RoboDK station: Additive-Manufacturing-and-Machining-with-ABB-IRB-120-3-0-6.rdk

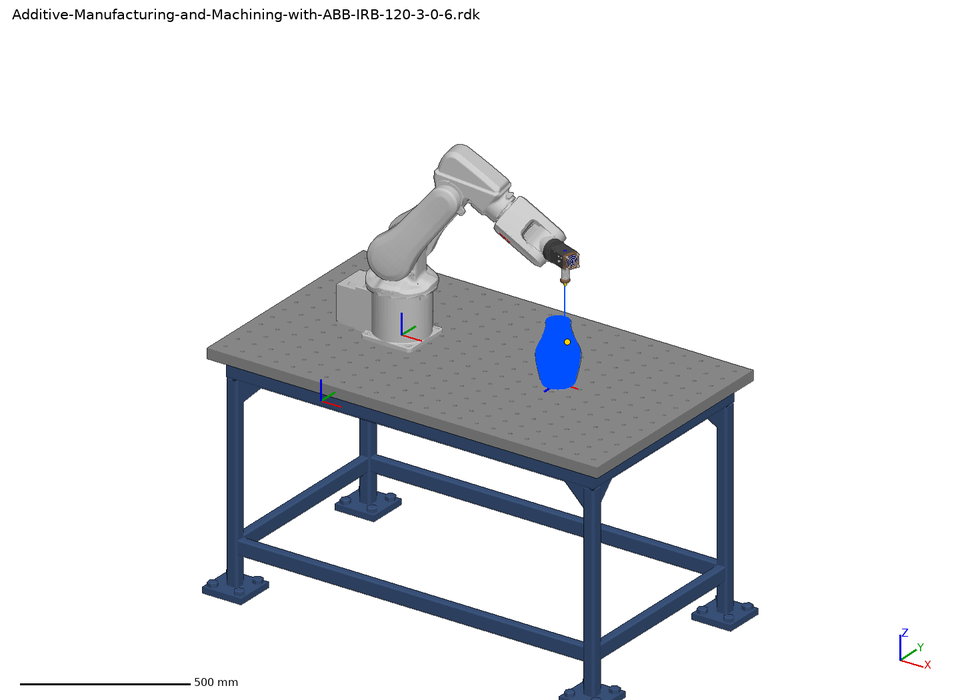
[picture v0: the station drawn from its stored meshes, robots at their saved joint values, targets as dots, program paths as lines]
Station Additive Manufacturing and Machining with ABB IRB 120-3/0.6 (saved by RoboDK 6.0.0). Poses are relative to the parent item; angles as X-Y-Z fixed-axis rotations.
Station parameters (name, value as stored): TAGS, ['Additive Manufacturing'], CEAD Extruder E40, 0
  - frame ABB IRB 120-3/0.6 Base at (-170, 0, 0) mm
    - robot ABB IRB 120-3/0.6: 6 axes, payload 3 kg, reach 580 mm, repeatability 0.01 mm, weight 25 kg
        modified DH rows (alpha deg, a mm, theta deg, d mm): 0, 0, 0, 290; -90, 0, -90, 0; 0, 270, 0, 0; -90, 70, 0, 302; 90, 0, 0, 0; -90, 0, 180, 72
        joint limits [-165, -110, -90, -160, -120, -400] to [165, 110, 70, 160, 120, 400]; home [0, 0, 0, 0, 0, 0]; saved at [10.704, 38.544, -4.293, -133.463, 44.707, 143.134]
      - tool ExtruderTool, TCP at (89.07, -8.14, 48.79) mm, rotated rx 0 ry 90 rz 0 deg, size 118.8 x 58.1 x 78.5 mm
    - object Table 1400x800x800mm at (-80, 0, 0) mm, size 1420 x 820 x 800 mm, geometry from UUID&
    - frame Part Reference at (560, 0, 0) mm, rotated rx 90 ry 0 rz 0 deg
      - object Simple Vase at (0, 0, 0) mm, size 135.9 x 200 x 135.9 mm, geometry from UUID&
      - frame NC File Frame at (-500, 0, 500) mm, rotated rx -90 ry 0 rz 0 deg
  - machining project Path1 settings: C:/Users/oli82/Desktop/List of demonstrations/8. G-code 3D printing/Vase.gcode | rotZ(0) | rotX(0)*rotY(0) | rotz(0)
  - program Path1 (30125 instructions, listed below)
  - Python program ExtrusionStart (listed below)
  - Python program ExtrusionStop (listed below)
  - notes Description: <!DOCTYPE HTML PUBLIC "-//W3C//DTD HTML 4.0//EN" "http://www.w3.org/TR/REC-html40/strict.dtd">
<html><head><meta name="qrichtext" content="1" /><style type="text/css">
p, li { white-space: pre-wrap; }
</style></head><body style=" font-family:'MS Shell Dlg 2'; font-size:8.25pt; font-weight:400; font-style:normal;">
<p style=" margin-top:0px; margin-bottom:0px; margin-left:0px; margin-right:0px; -qt-block-indent:0; text-indent:0px;">This example showcase the 3D printing of a vase using a ABB IRB 120-3/0.6 robot.<br /><br />Link for download : <a href="https://robodk.com/example/Additive-Manufacturing-and-Machining-with-ABB-IRB-120-3-0-6"><span style=" text-decoration: underline; color:#2a82da;">Additive Manufacturing and Machining with ABB IRB 120-3/0.6 robot | Examples Library</span></a></p></body></html>
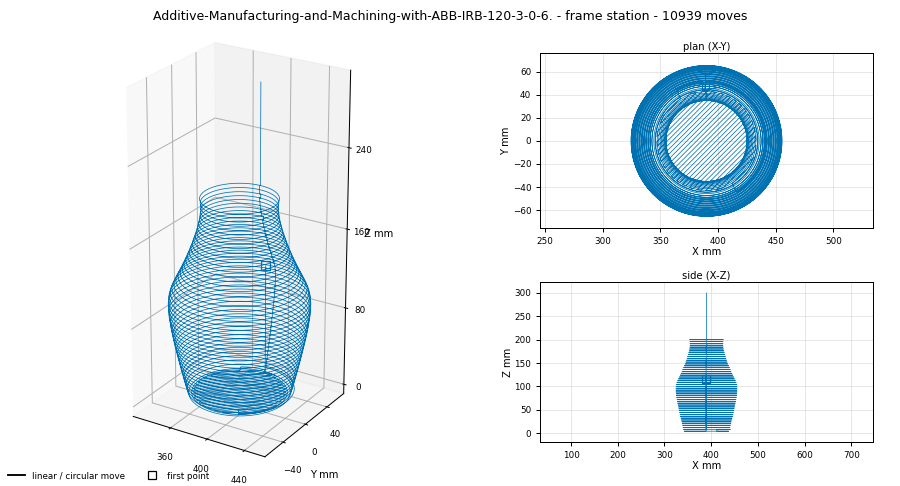
[picture p0: tool path of Additive-Manufacturing-and-Machining-with-ABB-IRB-120-3-0-6.rdk in frame station, 10939 of 10939 moves have a stored position in this frame; points joined in program order, loops and branches not executed]

--- program Path1 (robot ABB IRB 120-3/0.6) ---
  Smooth(1)
  Call SetRPM(200.0)
  Call M_RunCode(104)
  Call M_RunCode(105)
  Call SetRPM(200.0)
  Call M_RunCode(109)
  Call M_RunCode(82)
  Set speed (100.0 mm/s)
  Set speed (1000.0 mm/s)
  Set Ref.: NC File Frame
  Set Tool: ExtruderTool
  Show ExtruderTool
  MoveJ 1 to (499.11, 547.5, 115) mm, rotated rx 180 ry 0 rz 160 deg; joints [12.14, 61.149, -3.875, -143.247, 62.756, 161.126]
  MoveL 2 to (499.11, 547.5, 115) mm, rotated rx 180 ry 0 rz 160 deg; joints [12.14, 61.149, -3.875, -143.247, 62.756, 161.126]
  MoveL 3 to (499.11, 547.5, 15) mm, rotated rx -180 ry 0 rz 160 deg; joints [12.14, 78.131, -13.92, -145.093, 68.384, 165.584]
  Call ExtrusionStart
  MoveL 4 to (499.11, 547.5, 15) mm, rotated rx -180 ry 0 rz 160 deg; joints [12.14, 78.131, -13.92, -145.093, 68.384, 165.584]
  Call Extruder(0.00000)
  Set speed (3.3 mm/s)
  Call Extruder(3.00000)
  MoveL 5 to (499.11, 547.5, 15) mm, rotated rx -180 ry 0 rz 160 deg; joints [12.14, 78.131, -13.92, -145.093, 68.384, 165.584]
  Call Extruder(0.00000)
  Call Extruder(0.00000)
  Call Extruder(0.00000)
  Set speed (25.0 mm/s)
  Call Extruder(-6.50000)
  MoveL 6 to (499.11, 547.5, 15) mm, rotated rx -180 ry 0 rz 160 deg; joints [12.14, 78.131, -13.92, -145.093, 68.384, 165.584]
  Call M_RunCode(107)
  Set speed (60.0 mm/s)
  MoveL 7 to (499.11, 547.5, 4) mm, rotated rx 180 ry 0 rz 160 deg; joints [12.14, 80.192, -15.549, -145.19, 68.738, 165.849]
  Set speed (25.0 mm/s)
  Call Extruder(0.00000)
  MoveL 8 to (499.11, 547.5, 4) mm, rotated rx 180 ry 0 rz 160 deg; joints [12.14, 80.192, -15.549, -145.19, 68.738, 165.849]
  Set speed (30.0 mm/s)
  Call Extruder(3.94045)
  MoveL 9 to (497.01, 547.41, 4) mm, rotated rx 180 ry 0 rz 160 deg; joints [12.185, 79.885, -14.815, -145.238, 69.099, 166.093]
  Call Extruder(5.40756)
  MoveL 10 to (496.24, 547.36, 4) mm, rotated rx 180 ry 0 rz 160 deg; joints [12.199, 79.771, -14.543, -145.258, 69.233, 166.185]
  Call Extruder(7.73662)
  MoveL 11 to (495, 547.24, 4) mm, rotated rx -180 ry 0 rz 160 deg; joints [12.218, 79.591, -14.112, -145.292, 69.444, 166.331]
  Call Extruder(9.97998)
  MoveL 12 to (493.82, 547.1, 4) mm, rotated rx 180 ry 0 rz 160 deg; joints [12.232, 79.42, -13.698, -145.329, 69.647, 166.473]
  Call Extruder(11.58516)
  MoveL 13 to (492.97, 546.98, 4) mm, rotated rx 180 ry 0 rz 160 deg; joints [12.24, 79.297, -13.403, -145.357, 69.791, 166.575]
  Call Extruder(13.82687)
  MoveL 14 to (491.8, 546.79, 4) mm, rotated rx -180 ry 0 rz 160 deg; joints [12.247, 79.128, -12.992, -145.399, 69.991, 166.718]
  Call Extruder(15.46933)
  MoveL 15 to (490.94, 546.63, 4) mm, rotated rx 180 ry 0 rz 160 deg; joints [12.25, 79.004, -12.693, -145.433, 70.137, 166.824]
  Call Extruder(17.73552)
  MoveL 16 to (489.76, 546.39, 4) mm, rotated rx -180 ry 0 rz 160 deg; joints [12.253, 78.835, -12.282, -145.48, 70.337, 166.969]
  Call Extruder(20.50129)
  MoveL 17 to (488.33, 546.05, 4) mm, rotated rx 180 ry 0 rz 160 deg; joints [12.249, 78.631, -11.783, -145.543, 70.578, 167.147]
  Call Extruder(21.54013)
  MoveL 18 to (487.79, 545.91, 4) mm, rotated rx -180 ry 0 rz 160 deg; joints [12.246, 78.555, -11.597, -145.567, 70.668, 167.214]
  Call Extruder(24.36141)
  MoveL 19 to (486.35, 545.5, 4) mm, rotated rx -180 ry 0 rz 160 deg; joints [12.234, 78.35, -11.095, -145.638, 70.911, 167.396]
  Call Extruder(25.41345)
  MoveL 20 to (485.82, 545.34, 4) mm, rotated rx 180 ry 0 rz 160 deg; joints [12.228, 78.275, -10.909, -145.666, 71.001, 167.464]
  Call Extruder(29.35669)
  MoveL 21 to (483.83, 544.67, 4) mm, rotated rx 180 ry 0 rz 160 deg; joints [12.198, 77.995, -10.217, -145.776, 71.334, 167.719]
  Call Extruder(30.41593)
  MoveL 22 to (483.3, 544.47, 4) mm, rotated rx -180 ry 0 rz 160 deg; joints [12.188, 77.921, -10.033, -145.807, 71.423, 167.787]
  Call Extruder(33.18350)
  MoveL 23 to (481.93, 543.94, 4) mm, rotated rx -180 ry 0 rz 160 deg; joints [12.157, 77.729, -9.557, -145.893, 71.652, 167.966]
  Call Extruder(34.27379)
  MoveL 24 to (481.4, 543.71, 4) mm, rotated rx -180 ry 0 rz 160 deg; joints [12.143, 77.654, -9.371, -145.927, 71.742, 168.036]
  Call Extruder(36.99791)
  MoveL 25 to (480.07, 543.12, 4) mm, rotated rx 180 ry 0 rz 160 deg; joints [12.104, 77.469, -8.91, -146.018, 71.962, 168.211]
  Call Extruder(38.43745)
  MoveL 26 to (479.38, 542.79, 4) mm, rotated rx 180 ry 0 rz 160 deg; joints [12.081, 77.373, -8.669, -146.068, 72.078, 168.303]
  Call Extruder(38.46458)
  MoveL 27 to (479.37, 542.8, 4) mm, rotated rx 180 ry 0 rz 160 deg; joints [12.082, 77.372, -8.666, -146.067, 72.08, 168.304]
  Call Extruder(42.05595)
  MoveL 28 to (477.67, 541.93, 4) mm, rotated rx -180 ry 0 rz 160 deg; joints [12.018, 77.136, -8.073, -146.198, 72.363, 168.533]
  Call Extruder(43.31085)
  MoveL 29 to (477.08, 541.61, 4) mm, rotated rx 180 ry 0 rz 160 deg; joints [11.993, 77.055, -7.868, -146.245, 72.461, 168.613]
  Call Extruder(45.90183)
  MoveL 30 to (475.89, 540.93, 4) mm, rotated rx 180 ry 0 rz 160 deg; joints [11.937, 76.889, -7.451, -146.346, 72.66, 168.777]
  Call Extruder(47.00351)
  MoveL 31 to (475.39, 540.63, 4) mm, rotated rx -180 ry 0 rz 160 deg; joints [11.912, 76.82, -7.275, -146.39, 72.744, 168.846]
  Call Extruder(50.33195)
  MoveL 32 to (473.88, 539.69, 4) mm, rotated rx -180 ry 0 rz 160 deg; joints [11.832, 76.614, -6.75, -146.527, 72.993, 169.055]
  Call Extruder(53.58788)
  MoveL 33 to (472.46, 538.71, 4) mm, rotated rx 180 ry 0 rz 160 deg; joints [11.743, 76.418, -6.25, -146.669, 73.231, 169.256]
  Call Extruder(55.85392)
  MoveL 34 to (471.49, 538, 4) mm, rotated rx 180 ry 0 rz 160 deg; joints [11.676, 76.285, -5.909, -146.772, 73.392, 169.395]
  Call Extruder(58.62690)
  MoveL 35 to (470.32, 537.09, 4) mm, rotated rx 180 ry 0 rz 160 deg; joints [11.589, 76.125, -5.498, -146.902, 73.587, 169.564]
  Call Extruder(59.70505)
  MoveL 36 to (469.88, 536.73, 4) mm, rotated rx -180 ry 0 rz 160 deg; joints [11.554, 76.064, -5.341, -146.953, 73.661, 169.629]
  Call Extruder(62.48300)
  MoveL 37 to (468.75, 535.78, 4) mm, rotated rx 180 ry 0 rz 160 deg; joints [11.459, 75.91, -4.942, -147.089, 73.849, 169.794]
  Call Extruder(63.55306)
  MoveL 38 to (468.32, 535.4, 4) mm, rotated rx 180 ry 0 rz 160 deg; joints [11.421, 75.852, -4.791, -147.143, 73.92, 169.858]
  Call Extruder(66.33620)
  MoveL 39 to (467.24, 534.4, 4) mm, rotated rx 180 ry 0 rz 160 deg; joints [11.317, 75.703, -4.406, -147.286, 74.101, 170.021]
  Call Extruder(68.54172)
  MoveL 40 to (466.4, 533.58, 4) mm, rotated rx -180 ry 0 rz 160 deg; joints [11.23, 75.588, -4.106, -147.403, 74.242, 170.148]
  Call Extruder(71.29259)
  MoveL 41 to (465.38, 532.53, 4) mm, rotated rx -180 ry 0 rz 160 deg; joints [11.118, 75.449, -3.741, -147.552, 74.413, 170.305]
  Call Extruder(75.20093)
  MoveL 42 to (463.99, 530.99, 4) mm, rotated rx 180 ry 0 rz 160 deg; joints [10.948, 75.259, -3.242, -147.772, 74.646, 170.523]
  Call Extruder(76.26841)
  MoveL 43 to (463.62, 530.55, 4) mm, rotated rx 180 ry 0 rz 160 deg; joints [10.9, 75.209, -3.109, -147.833, 74.708, 170.582]
  Call Extruder(79.02172)
  MoveL 44 to (462.7, 529.42, 4) mm, rotated rx -180 ry 0 rz 160 deg; joints [10.771, 75.082, -2.774, -147.995, 74.863, 170.731]
  Call Extruder(81.24900)
  MoveL 45 to (461.98, 528.48, 4) mm, rotated rx -180 ry 0 rz 160 deg; joints [10.663, 74.983, -2.512, -148.128, 74.985, 170.849]
  Call Extruder(84.79388)
  MoveL 46 to (460.88, 526.95, 4) mm, rotated rx -180 ry 0 rz 160 deg; joints [10.485, 74.83, -2.107, -148.346, 75.171, 171.034]
  Call Extruder(87.90382)
  MoveL 47 to (459.96, 525.57, 4) mm, rotated rx 180 ry 0 rz 160 deg; joints [10.321, 74.704, -1.769, -148.543, 75.326, 171.191]
  Call Extruder(88.98138)
  MoveL 48 to (459.66, 525.09, 4) mm, rotated rx -180 ry 0 rz 160 deg; joints [10.263, 74.661, -1.654, -148.612, 75.379, 171.245]
  Call Extruder(91.75605)
  MoveL 49 to (458.9, 523.82, 4) mm, rotated rx 180 ry 0 rz 160 deg; joints [10.11, 74.555, -1.37, -148.792, 75.508, 171.38]
  Call Extruder(92.84401)
  MoveL 50 to (458.61, 523.32, 4) mm, rotated rx -180 ry 0 rz 160 deg; joints [10.048, 74.514, -1.261, -148.864, 75.557, 171.432]
  Call Extruder(95.61321)
  MoveL 51 to (457.91, 522.03, 4) mm, rotated rx -180 ry 0 rz 160 deg; joints [9.889, 74.415, -0.993, -149.049, 75.678, 171.562]
  Call Extruder(97.83579)
  MoveL 52 to (457.37, 520.97, 4) mm, rotated rx -180 ry 0 rz 160 deg; joints [9.757, 74.339, -0.787, -149.2, 75.77, 171.664]
  Call Extruder(100.62179)
  MoveL 53 to (456.74, 519.63, 4) mm, rotated rx -180 ry 0 rz 160 deg; joints [9.589, 74.248, -0.541, -149.393, 75.879, 171.788]
  Call Extruder(101.67932)
  MoveL 54 to (456.51, 519.12, 4) mm, rotated rx 180 ry 0 rz 160 deg; joints [9.523, 74.214, -0.45, -149.466, 75.919, 171.834]
  Call Extruder(104.48226)
  MoveL 55 to (455.93, 517.75, 4) mm, rotated rx 180 ry 0 rz 160 deg; joints [9.348, 74.13, -0.22, -149.664, 76.02, 171.953]
  Call Extruder(105.53437)
  MoveL 56 to (455.73, 517.23, 4) mm, rotated rx 180 ry 0 rz 160 deg; joints [9.281, 74.099, -0.137, -149.739, 76.056, 171.997]
  Call Extruder(109.42611)
  MoveL 57 to (455.02, 515.28, 4) mm, rotated rx -180 ry 0 rz 160 deg; joints [9.028, 73.993, 0.153, -150.019, 76.18, 172.154]
  Call Extruder(112.17917)
  MoveL 58 to (454.57, 513.89, 4) mm, rotated rx -180 ry 0 rz 160 deg; joints [8.845, 73.923, 0.343, -150.221, 76.259, 172.26]
  Call Extruder(114.41161)
  MoveL 59 to (454.24, 512.75, 4) mm, rotated rx 180 ry 0 rz 160 deg; joints [8.694, 73.871, 0.486, -150.386, 76.318, 172.343]
  Call Extruder(117.17477)
  MoveL 60 to (453.86, 511.33, 4) mm, rotated rx 180 ry 0 rz 160 deg; joints [8.505, 73.81, 0.653, -150.591, 76.386, 172.442]
  Call Extruder(118.23559)
  MoveL 61 to (453.73, 510.78, 4) mm, rotated rx -180 ry 0 rz 160 deg; joints [8.431, 73.789, 0.713, -150.671, 76.409, 172.479]
  Call Extruder(121.02778)
  MoveL 62 to (453.42, 509.33, 4) mm, rotated rx -180 ry 0 rz 160 deg; joints [8.236, 73.735, 0.861, -150.882, 76.466, 172.573]
  Call Extruder(123.26684)
  MoveL 63 to (453.2, 508.16, 4) mm, rotated rx 180 ry 0 rz 160 deg; joints [8.077, 73.695, 0.97, -151.052, 76.506, 172.646]
  Call Extruder(124.88048)
  MoveL 64 to (453.06, 507.31, 4) mm, rotated rx 180 ry 0 rz 160 deg; joints [7.962, 73.668, 1.043, -151.175, 76.533, 172.696]
  Call Extruder(127.12304)
  MoveL 65 to (452.89, 506.13, 4) mm, rotated rx 180 ry 0 rz 160 deg; joints [7.8, 73.635, 1.137, -151.347, 76.565, 172.764]
  Call Extruder(128.72549)
  MoveL 66 to (452.79, 505.29, 4) mm, rotated rx 180 ry 0 rz 160 deg; joints [7.684, 73.613, 1.198, -151.47, 76.584, 172.811]
  Call Extruder(130.96145)
  MoveL 67 to (452.68, 504.11, 4) mm, rotated rx 180 ry 0 rz 160 deg; joints [7.52, 73.585, 1.275, -151.642, 76.607, 172.874]
  Call Extruder(134.81308)
  MoveL 68 to (452.54, 502.06, 4) mm, rotated rx -180 ry 0 rz 160 deg; joints [7.236, 73.544, 1.388, -151.94, 76.635, 172.976]
  Call Extruder(138.66641)
  MoveL 69 to (452.49, 500.01, 4) mm, rotated rx 180 ry 0 rz 160 deg; joints [6.949, 73.514, 1.472, -152.238, 76.648, 173.069]
  Call Extruder(142.35037)
  MoveL 70 to (452.54, 498.06, 4) mm, rotated rx -180 ry 0 rz 160 deg; joints [6.673, 73.494, 1.526, -152.524, 76.646, 173.151]
  Call Extruder(145.97620)
  MoveL 71 to (452.65, 496.13, 4) mm, rotated rx 180 ry 0 rz 160 deg; joints [6.401, 73.484, 1.555, -152.804, 76.63, 173.224]
  Call Extruder(148.37186)
  MoveL 72 to (452.77, 494.86, 4) mm, rotated rx -180 ry 0 rz 160 deg; joints [6.22, 73.482, 1.561, -152.989, 76.612, 173.268]
  Call Extruder(151.58092)
  MoveL 73 to (452.99, 493.17, 4) mm, rotated rx 180 ry 0 rz 160 deg; joints [5.979, 73.485, 1.55, -153.235, 76.578, 173.322]
  Call Extruder(155.28658)
  MoveL 74 to (453.31, 491.23, 4) mm, rotated rx 180 ry 0 rz 160 deg; joints [5.7, 73.498, 1.515, -153.517, 76.525, 173.378]
  Call Extruder(158.89603)
  MoveL 75 to (453.7, 489.35, 4) mm, rotated rx 180 ry 0 rz 160 deg; joints [5.43, 73.519, 1.457, -153.789, 76.461, 173.425]
  Call Extruder(160.89432)
  MoveL 76 to (453.96, 488.32, 4) mm, rotated rx 180 ry 0 rz 160 deg; joints [5.281, 73.535, 1.413, -153.938, 76.419, 173.448]
  Call Extruder(162.51775)
  MoveL 77 to (454.18, 487.48, 4) mm, rotated rx 180 ry 0 rz 160 deg; joints [5.161, 73.55, 1.372, -154.058, 76.381, 173.465]
  Call Extruder(164.55536)
  MoveL 78 to (454.47, 486.44, 4) mm, rotated rx -180 ry 0 rz 160 deg; joints [5.011, 73.57, 1.315, -154.208, 76.331, 173.485]
  Call Extruder(168.16278)
  MoveL 79 to (455.06, 484.62, 4) mm, rotated rx -180 ry 0 rz 160 deg; joints [4.746, 73.614, 1.194, -154.47, 76.232, 173.515]
  Call Extruder(171.85348)
  MoveL 80 to (455.73, 482.77, 4) mm, rotated rx 180 ry 0 rz 160 deg; joints [4.479, 73.668, 1.045, -154.733, 76.116, 173.538]
  Call Extruder(175.47423)
  MoveL 81 to (456.46, 480.99, 4) mm, rotated rx 180 ry 0 rz 160 deg; joints [4.222, 73.729, 0.875, -154.986, 75.989, 173.555]
  Call Extruder(177.47050)
  MoveL 82 to (456.9, 480.02, 4) mm, rotated rx -180 ry 0 rz 160 deg; joints [4.081, 73.767, 0.772, -155.122, 75.914, 173.561]
  Call Extruder(179.11206)
  MoveL 83 to (457.27, 479.24, 4) mm, rotated rx 180 ry 0 rz 160 deg; joints [3.967, 73.8, 0.681, -155.233, 75.848, 173.564]
  Call Extruder(181.39349)
  MoveL 84 to (457.81, 478.15, 4) mm, rotated rx 180 ry 0 rz 160 deg; joints [3.81, 73.849, 0.548, -155.386, 75.754, 173.567]
  Call Extruder(181.42382)
  MoveL 85 to (457.83, 478.14, 4) mm, rotated rx 180 ry 0 rz 160 deg; joints [3.808, 73.85, 0.544, -155.387, 75.751, 173.567]
  Call Extruder(184.79550)
  MoveL 86 to (458.68, 476.57, 4) mm, rotated rx 180 ry 0 rz 160 deg; joints [3.58, 73.928, 0.329, -155.607, 75.602, 173.566]
  Call Extruder(188.39318)
  MoveL 87 to (459.65, 474.92, 4) mm, rotated rx -180 ry 0 rz 160 deg; joints [3.342, 74.02, 0.079, -155.834, 75.43, 173.56]
  Call Extruder(190.39943)
  MoveL 88 to (460.23, 474.02, 4) mm, rotated rx 180 ry 0 rz 160 deg; joints [3.212, 74.075, -0.073, -155.957, 75.328, 173.553]
  Call Extruder(192.01934)
  MoveL 89 to (460.71, 473.31, 4) mm, rotated rx -180 ry 0 rz 160 deg; joints [3.108, 74.122, -0.199, -156.055, 75.244, 173.547]
  Call Extruder(194.06074)
  MoveL 90 to (461.33, 472.42, 4) mm, rotated rx 180 ry 0 rz 160 deg; joints [2.98, 74.183, -0.364, -156.176, 75.133, 173.537]
  Call Extruder(195.68505)
  MoveL 91 to (461.84, 471.72, 4) mm, rotated rx -180 ry 0 rz 160 deg; joints [2.879, 74.233, -0.5, -156.271, 75.043, 173.527]
  Call Extruder(197.64737)
  MoveL 92 to (462.46, 470.88, 4) mm, rotated rx 180 ry 0 rz 160 deg; joints [2.759, 74.296, -0.671, -156.383, 74.932, 173.515]
  Call Extruder(201.35720)
  MoveL 93 to (463.71, 469.35, 4) mm, rotated rx 180 ry 0 rz 160 deg; joints [2.538, 74.422, -1.011, -156.586, 74.71, 173.486]
  Call Extruder(204.96266)
  MoveL 94 to (464.97, 467.91, 4) mm, rotated rx 180 ry 0 rz 160 deg; joints [2.332, 74.552, -1.363, -156.775, 74.484, 173.451]
  Call Extruder(206.96665)
  MoveL 95 to (465.7, 467.14, 4) mm, rotated rx 180 ry 0 rz 160 deg; joints [2.221, 74.629, -1.568, -156.875, 74.352, 173.429]
  Call Extruder(208.59616)
  MoveL 96 to (466.31, 466.52, 4) mm, rotated rx -180 ry 0 rz 160 deg; joints [2.132, 74.693, -1.739, -156.955, 74.244, 173.411]
  Call Extruder(210.62728)
  MoveL 97 to (467.08, 465.76, 4) mm, rotated rx -180 ry 0 rz 160 deg; joints [2.024, 74.774, -1.957, -157.051, 74.106, 173.386]
  Call Extruder(214.23995)
  MoveL 98 to (468.49, 464.45, 4) mm, rotated rx -180 ry 0 rz 160 deg; joints [1.839, 74.926, -2.362, -157.215, 73.852, 173.336]
  Call Extruder(217.86902)
  MoveL 99 to (469.95, 463.2, 4) mm, rotated rx -180 ry 0 rz 160 deg; joints [1.661, 75.086, -2.787, -157.369, 73.587, 173.281]
  Call Extruder(221.58056)
  MoveL 100 to (471.51, 461.99, 4) mm, rotated rx -180 ry 0 rz 160 deg; joints [1.49, 75.259, -3.242, -157.514, 73.305, 173.219]
  Call Extruder(223.56820)
  MoveL 101 to (472.36, 461.37, 4) mm, rotated rx 180 ry 0 rz 160 deg; joints [1.402, 75.355, -3.494, -157.587, 73.151, 173.183]
  Call Extruder(225.18427)
  MoveL 102 to (473.07, 460.87, 4) mm, rotated rx -180 ry 0 rz 160 deg; joints [1.333, 75.434, -3.703, -157.643, 73.023, 173.152]
  Call Extruder(227.15639)
  MoveL 103 to (473.94, 460.29, 4) mm, rotated rx 180 ry 0 rz 160 deg; joints [1.251, 75.533, -3.961, -157.71, 72.865, 173.114]
  Call Extruder(230.80766)
  MoveL 104 to (475.58, 459.25, 4) mm, rotated rx 180 ry 0 rz 160 deg; joints [1.107, 75.722, -4.455, -157.824, 72.566, 173.038]
  Call Extruder(234.46092)
  MoveL 105 to (477.27, 458.29, 4) mm, rotated rx -180 ry 0 rz 160 deg; joints [0.973, 75.919, -4.965, -157.926, 72.259, 172.956]
  Call Extruder(236.48707)
  MoveL 106 to (478.22, 457.79, 4) mm, rotated rx 180 ry 0 rz 160 deg; joints [0.904, 76.031, -5.256, -157.977, 72.085, 172.908]
  Call Extruder(238.11490)
  MoveL 107 to (478.99, 457.4, 4) mm, rotated rx 180 ry 0 rz 160 deg; joints [0.85, 76.123, -5.492, -158.016, 71.945, 172.868]
  Call Extruder(239.70662)
  MoveL 108 to (479.75, 457.03, 4) mm, rotated rx 180 ry 0 rz 160 deg; joints [0.799, 76.214, -5.726, -158.051, 71.805, 172.828]
  Call Extruder(241.75907)
  MoveL 109 to (480.74, 456.58, 4) mm, rotated rx 180 ry 0 rz 160 deg; joints [0.737, 76.333, -6.033, -158.093, 71.624, 172.775]
  Call Extruder(243.71701)
  MoveL 110 to (481.7, 456.16, 4) mm, rotated rx 180 ry 0 rz 160 deg; joints [0.68, 76.449, -6.329, -158.13, 71.449, 172.722]
  Call Extruder(247.36729)
  MoveL 111 to (483.5, 455.45, 4) mm, rotated rx -180 ry 0 rz 160 deg; joints [0.584, 76.67, -6.894, -158.188, 71.118, 172.62]
  Call Extruder(250.65225)
  MoveL 112 to (485.15, 454.88, 4) mm, rotated rx 180 ry 0 rz 160 deg; joints [0.506, 76.875, -7.414, -158.229, 70.815, 172.523]
  Call Extruder(250.68199)
  MoveL 113 to (485.16, 454.87, 4) mm, rotated rx 180 ry 0 rz 160 deg; joints [0.504, 76.876, -7.417, -158.23, 70.813, 172.523]
  Call Extruder(253.05781)
  MoveL 114 to (486.37, 454.49, 4) mm, rotated rx 180 ry 0 rz 160 deg; joints [0.454, 77.028, -7.8, -158.253, 70.592, 172.449]
  Call Extruder(254.66679)
  MoveL 115 to (487.19, 454.25, 4) mm, rotated rx 180 ry 0 rz 160 deg; joints [0.422, 77.132, -8.062, -158.266, 70.441, 172.399]
  Call Extruder(256.67033)
  MoveL 116 to (488.22, 453.98, 4) mm, rotated rx 180 ry 0 rz 160 deg; joints [0.385, 77.263, -8.392, -158.279, 70.251, 172.334]
  Call Extruder(260.34428)
  MoveL 117 to (490.12, 453.53, 4) mm, rotated rx -180 ry 0 rz 160 deg; joints [0.325, 77.507, -9.005, -158.292, 69.901, 172.21]
  Call Extruder(263.95004)
  MoveL 118 to (492.01, 453.17, 4) mm, rotated rx 180 ry 0 rz 160 deg; joints [0.276, 77.753, -9.618, -158.294, 69.553, 172.083]
  Call Extruder(267.62543)
  MoveL 119 to (493.94, 452.89, 4) mm, rotated rx 180 ry 0 rz 160 deg; joints [0.238, 78.009, -10.253, -158.281, 69.195, 171.947]
  Call Extruder(269.20801)
  MoveL 120 to (494.77, 452.78, 4) mm, rotated rx -180 ry 0 rz 160 deg; joints [0.225, 78.121, -10.53, -158.272, 69.041, 171.887]
  Call Extruder(273.22649)
  MoveL 121 to (496.9, 452.6, 4) mm, rotated rx -180 ry 0 rz 160 deg; joints [0.199, 78.409, -11.239, -158.239, 68.646, 171.73]
  Call Extruder(276.93202)
  MoveL 122 to (498.87, 452.51, 4) mm, rotated rx -180 ry 0 rz 160 deg; joints [0.187, 78.68, -11.901, -158.194, 68.28, 171.578]
  Call Extruder(280.53803)
  MoveL 123 to (500.79, 452.5, 4) mm, rotated rx 180 ry 0 rz 160 deg; joints [0.186, 78.947, -12.553, -158.138, 67.923, 171.424]
  Call Extruder(282.54608)
  MoveL 124 to (501.85, 452.53, 4) mm, rotated rx -180 ry 0 rz 160 deg; joints [0.189, 79.097, -12.919, -158.102, 67.724, 171.336]
  Call Extruder(284.19577)
  MoveL 125 to (502.73, 452.58, 4) mm, rotated rx -180 ry 0 rz 160 deg; joints [0.194, 79.222, -13.22, -158.069, 67.56, 171.263]
  Call Extruder(286.19216)
  MoveL 126 to (503.79, 452.65, 4) mm, rotated rx -180 ry 0 rz 160 deg; joints [0.203, 79.374, -13.587, -158.027, 67.362, 171.173]
  Call Extruder(289.85662)
  MoveL 127 to (505.73, 452.84, 4) mm, rotated rx 180 ry 0 rz 160 deg; joints [0.227, 79.654, -14.263, -157.939, 67, 171.002]
  Call Extruder(293.44499)
  MoveL 128 to (507.62, 453.11, 4) mm, rotated rx -180 ry 0 rz 160 deg; joints [0.259, 79.932, -14.929, -157.841, 66.645, 170.829]
  Call Extruder(297.15517)
  MoveL 129 to (509.56, 453.47, 4) mm, rotated rx -180 ry 0 rz 160 deg; joints [0.303, 80.222, -15.62, -157.729, 66.28, 170.645]
  Call Extruder(299.11774)
  MoveL 130 to (510.57, 453.69, 4) mm, rotated rx -180 ry 0 rz 160 deg; joints [0.33, 80.376, -15.986, -157.664, 66.089, 170.545]
  Call Extruder(300.75071)
  MoveL 131 to (511.42, 453.89, 4) mm, rotated rx 180 ry 0 rz 160 deg; joints [0.354, 80.505, -16.292, -157.608, 65.929, 170.461]
  Call Extruder(302.73079)
  MoveL 132 to (512.44, 454.15, 4) mm, rotated rx -180 ry 0 rz 160 deg; joints [0.386, 80.661, -16.662, -157.537, 65.737, 170.357]
  Call Extruder(306.43685)
  MoveL 133 to (514.33, 454.71, 4) mm, rotated rx 180 ry 0 rz 160 deg; joints [0.453, 80.955, -17.356, -157.395, 65.379, 170.159]
  Call Extruder(310.02735)
  MoveL 134 to (516.14, 455.32, 4) mm, rotated rx 180 ry 0 rz 160 deg; joints [0.526, 81.241, -18.026, -157.246, 65.036, 169.962]
  Call Extruder(313.68619)
  MoveL 135 to (517.95, 456.02, 4) mm, rotated rx -180 ry 0 rz 160 deg; joints [0.61, 81.532, -18.708, -157.084, 64.692, 169.756]
  Call Extruder(316.29999)
  MoveL 136 to (519.23, 456.56, 4) mm, rotated rx -180 ry 0 rz 160 deg; joints [0.674, 81.741, -19.194, -156.963, 64.448, 169.606]
  Call Extruder(319.28823)
  MoveL 137 to (520.67, 457.23, 4) mm, rotated rx 180 ry 0 rz 160 deg; joints [0.754, 81.978, -19.745, -156.816, 64.173, 169.432]
  Call Extruder(322.97713)
  MoveL 138 to (522.42, 458.12, 4) mm, rotated rx -180 ry 0 rz 160 deg; joints [0.859, 82.271, -20.423, -156.627, 63.839, 169.212]
  Call Extruder(326.64168)
  MoveL 139 to (524.12, 459.07, 4) mm, rotated rx -180 ry 0 rz 160 deg; joints [0.972, 82.56, -21.09, -156.429, 63.514, 168.99]
  Call Extruder(328.60959)
  MoveL 140 to (525.01, 459.62, 4) mm, rotated rx -180 ry 0 rz 160 deg; joints [1.036, 82.714, -21.444, -156.319, 63.343, 168.868]
  Call Extruder(330.23683)
  MoveL 141 to (525.74, 460.08, 4) mm, rotated rx -180 ry 0 rz 160 deg; joints [1.09, 82.842, -21.737, -156.226, 63.202, 168.767]
  Call Extruder(332.28040)
  MoveL 142 to (526.65, 460.68, 4) mm, rotated rx -180 ry 0 rz 160 deg; joints [1.16, 83.001, -22.102, -156.107, 63.028, 168.639]
  Call Extruder(335.86729)
  MoveL 143 to (528.21, 461.77, 4) mm, rotated rx 180 ry 0 rz 160 deg; joints [1.288, 83.279, -22.736, -155.892, 62.728, 168.412]
  Call Extruder(339.56123)
  MoveL 144 to (529.76, 462.97, 4) mm, rotated rx 180 ry 0 rz 160 deg; joints [1.427, 83.561, -23.378, -155.662, 62.428, 168.175]
  Call Extruder(343.17226)
  MoveL 145 to (531.23, 464.21, 4) mm, rotated rx 180 ry 0 rz 160 deg; joints [1.57, 83.832, -23.993, -155.429, 62.144, 167.941]
  Call Extruder(345.20914)
  MoveL 146 to (532.04, 464.93, 4) mm, rotated rx -180 ry 0 rz 160 deg; joints [1.653, 83.983, -24.335, -155.295, 61.988, 167.808]
  Call Extruder(346.80624)
  MoveL 147 to (532.66, 465.51, 4) mm, rotated rx 180 ry 0 rz 160 deg; joints [1.72, 84.1, -24.6, -155.188, 61.868, 167.703]
  Call Extruder(348.81641)
  MoveL 148 to (533.43, 466.25, 4) mm, rotated rx 180 ry 0 rz 160 deg; joints [1.805, 84.247, -24.931, -155.052, 61.719, 167.57]
  Call Extruder(351.57520)
  MoveL 149 to (534.46, 467.3, 4) mm, rotated rx -180 ry 0 rz 160 deg; joints [1.925, 84.445, -25.377, -154.862, 61.521, 167.388]
  Call Extruder(352.64929)
  MoveL 150 to (534.85, 467.72, 4) mm, rotated rx 180 ry 0 rz 160 deg; joints [1.973, 84.521, -25.548, -154.787, 61.445, 167.316]
  Call Extruder(355.43712)
  MoveL 151 to (535.84, 468.82, 4) mm, rotated rx 180 ry 0 rz 160 deg; joints [2.099, 84.717, -25.987, -154.59, 61.253, 167.131]
  Call Extruder(357.66289)
  MoveL 152 to (536.6, 469.72, 4) mm, rotated rx 180 ry 0 rz 160 deg; joints [2.201, 84.87, -26.33, -154.431, 61.105, 166.982]
  Call Extruder(360.42699)
  MoveL 153 to (537.52, 470.87, 4) mm, rotated rx -180 ry 0 rz 160 deg; joints [2.332, 85.057, -26.748, -154.231, 60.926, 166.798]
  Call Extruder(361.48983)
  MoveL 154 to (537.87, 471.31, 4) mm, rotated rx -180 ry 0 rz 160 deg; joints [2.383, 85.127, -26.905, -154.153, 60.86, 166.727]
  Call Extruder(364.29245)
  MoveL 155 to (538.75, 472.52, 4) mm, rotated rx 180 ry 0 rz 160 deg; joints [2.52, 85.31, -27.311, -153.945, 60.69, 166.54]
  Call Extruder(365.39196)
  MoveL 156 to (539.08, 473, 4) mm, rotated rx 180 ry 0 rz 160 deg; joints [2.574, 85.38, -27.468, -153.864, 60.626, 166.467]
  Call Extruder(368.17216)
  MoveL 157 to (539.9, 474.23, 4) mm, rotated rx -180 ry 0 rz 160 deg; joints [2.713, 85.554, -27.855, -153.655, 60.467, 166.282]
  Call Extruder(369.25694)
  MoveL 158 to (540.21, 474.71, 4) mm, rotated rx 180 ry 0 rz 160 deg; joints [2.768, 85.621, -28.004, -153.573, 60.407, 166.21]
  Call Extruder(372.02874)
  MoveL 159 to (540.98, 475.97, 4) mm, rotated rx 180 ry 0 rz 160 deg; joints [2.911, 85.788, -28.372, -153.362, 60.26, 166.027]
  Call Extruder(374.20232)
  MoveL 160 to (541.55, 476.98, 4) mm, rotated rx 180 ry 0 rz 160 deg; joints [3.024, 85.914, -28.652, -153.196, 60.151, 165.885]
  Call Extruder(377.00133)
  MoveL 161 to (542.25, 478.29, 4) mm, rotated rx 180 ry 0 rz 160 deg; joints [3.172, 86.072, -29.001, -152.98, 60.017, 165.702]
  Call Extruder(378.06886)
  MoveL 162 to (542.51, 478.79, 4) mm, rotated rx 180 ry 0 rz 160 deg; joints [3.23, 86.13, -29.13, -152.898, 59.968, 165.633]
  Call Extruder(380.87971)
  MoveL 163 to (543.16, 480.14, 4) mm, rotated rx 180 ry 0 rz 160 deg; joints [3.382, 86.28, -29.461, -152.68, 59.845, 165.453]
  Call Extruder(381.93973)
  MoveL 164 to (543.39, 480.65, 4) mm, rotated rx 180 ry 0 rz 160 deg; joints [3.44, 86.335, -29.581, -152.597, 59.802, 165.385]
  Call Extruder(384.69644)
  MoveL 165 to (543.96, 482, 4) mm, rotated rx -180 ry 0 rz 160 deg; joints [3.592, 86.472, -29.883, -152.383, 59.694, 165.211]
  Call Extruder(386.92783)
  MoveL 166 to (544.4, 483.11, 4) mm, rotated rx 180 ry 0 rz 160 deg; joints [3.716, 86.578, -30.117, -152.209, 59.613, 165.072]
  Call Extruder(389.71983)
  MoveL 167 to (544.9, 484.5, 4) mm, rotated rx 180 ry 0 rz 160 deg; joints [3.873, 86.705, -30.395, -151.991, 59.52, 164.901]
  Call Extruder(390.77628)
  MoveL 168 to (545.08, 485.03, 4) mm, rotated rx 180 ry 0 rz 160 deg; joints [3.933, 86.751, -30.496, -151.908, 59.487, 164.837]
  Call Extruder(393.58547)
  MoveL 169 to (545.53, 486.46, 4) mm, rotated rx 180 ry 0 rz 160 deg; joints [4.094, 86.869, -30.753, -151.69, 59.406, 164.668]
  Call Extruder(394.67589)
  MoveL 170 to (545.7, 487.01, 4) mm, rotated rx -180 ry 0 rz 160 deg; joints [4.156, 86.912, -30.849, -151.605, 59.377, 164.604]
  Call Extruder(397.43358)
  MoveL 171 to (546.07, 488.43, 4) mm, rotated rx -180 ry 0 rz 160 deg; joints [4.316, 87.016, -31.076, -151.391, 59.311, 164.444]
  Call Extruder(398.50525)
  MoveL 172 to (546.21, 488.98, 4) mm, rotated rx 180 ry 0 rz 160 deg; joints [4.379, 87.055, -31.161, -151.308, 59.288, 164.383]
  Call Extruder(401.27005)
  MoveL 173 to (546.53, 490.42, 4) mm, rotated rx 180 ry 0 rz 160 deg; joints [4.541, 87.148, -31.364, -151.095, 59.235, 164.228]
  Call Extruder(403.50646)
  MoveL 174 to (546.75, 491.59, 4) mm, rotated rx -180 ry 0 rz 160 deg; joints [4.673, 87.217, -31.515, -150.923, 59.199, 164.107]
  Call Extruder(405.14021)
  MoveL 175 to (546.9, 492.44, 4) mm, rotated rx -180 ry 0 rz 160 deg; joints [4.769, 87.265, -31.619, -150.799, 59.177, 164.019]
  Call Extruder(407.33763)
  MoveL 176 to (547.07, 493.6, 4) mm, rotated rx -180 ry 0 rz 160 deg; joints [4.9, 87.324, -31.749, -150.632, 59.151, 163.904]
  Call Extruder(411.27865)
  MoveL 177 to (547.31, 495.68, 4) mm, rotated rx -180 ry 0 rz 160 deg; joints [5.136, 87.416, -31.949, -150.336, 59.123, 163.706]
  Call Extruder(415.08226)
  MoveL 178 to (547.45, 497.7, 4) mm, rotated rx 180 ry 0 rz 160 deg; joints [5.365, 87.489, -32.107, -150.054, 59.113, 163.525]
  Call Extruder(418.94179)
  MoveL 179 to (547.51, 499.75, 4) mm, rotated rx 180 ry 0 rz 160 deg; joints [5.599, 87.545, -32.23, -149.773, 59.123, 163.353]
  Call Extruder(422.87761)
  MoveL 180 to (547.47, 501.84, 4) mm, rotated rx 180 ry 0 rz 160 deg; joints [5.839, 87.583, -32.313, -149.493, 59.153, 163.189]
  Call Extruder(425.07382)
  MoveL 181 to (547.41, 503.01, 4) mm, rotated rx 180 ry 0 rz 160 deg; joints [5.972, 87.597, -32.342, -149.339, 59.178, 163.103]
  Call Extruder(426.66906)
  MoveL 182 to (547.35, 503.85, 4) mm, rotated rx 180 ry 0 rz 160 deg; joints [6.07, 87.603, -32.357, -149.228, 59.2, 163.043]
  Call Extruder(429.32430)
  MoveL 183 to (547.21, 505.26, 4) mm, rotated rx 180 ry 0 rz 160 deg; joints [6.232, 87.607, -32.364, -149.046, 59.243, 162.949]
  Call Extruder(432.82644)
  MoveL 184 to (546.97, 507.1, 4) mm, rotated rx 180 ry 0 rz 160 deg; joints [6.445, 87.599, -32.346, -148.812, 59.315, 162.833]
  Call Extruder(436.61784)
  MoveL 185 to (546.63, 509.09, 4) mm, rotated rx -180 ry 0 rz 160 deg; joints [6.676, 87.573, -32.29, -148.565, 59.409, 162.721]
  Call Extruder(440.56318)
  MoveL 186 to (546.18, 511.14, 4) mm, rotated rx 180 ry 0 rz 160 deg; joints [6.916, 87.528, -32.192, -148.316, 59.525, 162.618]
  Call Extruder(443.25130)
  MoveL 187 to (545.82, 512.52, 4) mm, rotated rx -180 ry 0 rz 160 deg; joints [7.078, 87.487, -32.103, -148.151, 59.615, 162.557]
  Call Extruder(445.47572)
  MoveL 188 to (545.5, 513.66, 4) mm, rotated rx 180 ry 0 rz 160 deg; joints [7.213, 87.446, -32.015, -148.017, 59.696, 162.511]
  Call Extruder(448.24205)
  MoveL 189 to (545.06, 515.06, 4) mm, rotated rx 180 ry 0 rz 160 deg; joints [7.379, 87.388, -31.888, -147.855, 59.804, 162.46]
  Call Extruder(449.31461)
  MoveL 190 to (544.87, 515.6, 4) mm, rotated rx -180 ry 0 rz 160 deg; joints [7.443, 87.363, -31.833, -147.793, 59.849, 162.443]
  Call Extruder(452.36793)
  MoveL 191 to (544.31, 517.12, 4) mm, rotated rx 180 ry 0 rz 160 deg; joints [7.625, 87.285, -31.664, -147.621, 59.981, 162.399]
  Call Extruder(452.39506)
  MoveL 192 to (544.32, 517.14, 4) mm, rotated rx 180 ry 0 rz 160 deg; joints [7.627, 87.287, -31.669, -147.618, 59.979, 162.397]
  Call Extruder(455.99859)
  MoveL 193 to (543.58, 518.9, 4) mm, rotated rx 180 ry 0 rz 160 deg; joints [7.84, 87.179, -31.432, -147.424, 60.152, 162.359]
  Call Extruder(458.19539)
  MoveL 194 to (543.1, 519.97, 4) mm, rotated rx -180 ry 0 rz 160 deg; joints [7.969, 87.108, -31.276, -147.308, 60.262, 162.341]
  Call Extruder(461.36134)
  MoveL 195 to (542.37, 521.49, 4) mm, rotated rx 180 ry 0 rz 160 deg; joints [8.154, 86.997, -31.035, -147.146, 60.428, 162.322]
  Call Extruder(464.83355)
  MoveL 196 to (541.5, 523.11, 4) mm, rotated rx 180 ry 0 rz 160 deg; joints [8.354, 86.862, -30.739, -146.976, 60.624, 162.315]
  Call Extruder(465.89514)
  MoveL 197 to (541.23, 523.6, 4) mm, rotated rx 180 ry 0 rz 160 deg; joints [8.415, 86.818, -30.642, -146.925, 60.687, 162.315]
  Call Extruder(468.70017)
  MoveL 198 to (540.47, 524.89, 4) mm, rotated rx 180 ry 0 rz 160 deg; joints [8.574, 86.698, -30.379, -146.795, 60.855, 162.32]
  Call Extruder(469.78008)
  MoveL 199 to (540.16, 525.37, 4) mm, rotated rx -180 ry 0 rz 160 deg; joints [8.635, 86.65, -30.273, -146.746, 60.922, 162.324]
  Call Extruder(472.56923)
  MoveL 200 to (539.35, 526.61, 4) mm, rotated rx 180 ry 0 rz 160 deg; joints [8.792, 86.519, -29.987, -146.623, 61.099, 162.339]
  Call Extruder(474.74456)
  MoveL 201 to (538.69, 527.57, 4) mm, rotated rx -180 ry 0 rz 160 deg; joints [8.912, 86.414, -29.754, -146.531, 61.242, 162.356]
  Call Extruder(477.55608)
  MoveL 202 to (537.8, 528.77, 4) mm, rotated rx 180 ry 0 rz 160 deg; joints [9.066, 86.27, -29.438, -146.415, 61.432, 162.384]
  Call Extruder(478.62455)
  MoveL 203 to (537.46, 529.22, 4) mm, rotated rx -180 ry 0 rz 160 deg; joints [9.125, 86.214, -29.315, -146.372, 61.506, 162.396]
  Call Extruder(481.38398)
  MoveL 204 to (536.54, 530.36, 4) mm, rotated rx 180 ry 0 rz 160 deg; joints [9.273, 86.064, -28.984, -146.266, 61.701, 162.434]
  Call Extruder(482.78118)
  MoveL 205 to (536.06, 530.93, 4) mm, rotated rx -180 ry 0 rz 160 deg; joints [9.347, 85.986, -28.811, -146.214, 61.803, 162.456]
  Call Extruder(485.29202)
  MoveL 206 to (535.17, 531.93, 4) mm, rotated rx 180 ry 0 rz 160 deg; joints [9.479, 85.842, -28.492, -146.124, 61.988, 162.499]
  Call Extruder(487.47771)
  MoveL 207 to (534.38, 532.78, 4) mm, rotated rx 180 ry 0 rz 160 deg; joints [9.592, 85.713, -28.207, -146.047, 62.151, 162.54]
  Call Extruder(490.24046)
  MoveL 208 to (533.36, 533.83, 4) mm, rotated rx -180 ry 0 rz 160 deg; joints [9.733, 85.545, -27.833, -145.956, 62.364, 162.599]
  Call Extruder(491.31936)
  MoveL 209 to (532.94, 534.23, 4) mm, rotated rx 180 ry 0 rz 160 deg; joints [9.787, 85.477, -27.683, -145.922, 62.448, 162.624]
  Call Extruder(494.12752)
  MoveL 210 to (531.85, 535.25, 4) mm, rotated rx 180 ry 0 rz 160 deg; joints [9.927, 85.299, -27.287, -145.835, 62.671, 162.693]
  Call Extruder(495.19742)
  MoveL 211 to (531.43, 535.62, 4) mm, rotated rx 180 ry 0 rz 160 deg; joints [9.979, 85.229, -27.132, -145.804, 62.757, 162.721]
  Call Extruder(497.97630)
  MoveL 212 to (530.3, 536.59, 4) mm, rotated rx -180 ry 0 rz 160 deg; joints [10.113, 85.046, -26.724, -145.725, 62.983, 162.798]
  Call Extruder(499.04861)
  MoveL 213 to (529.86, 536.95, 4) mm, rotated rx 180 ry 0 rz 160 deg; joints [10.164, 84.974, -26.563, -145.696, 63.071, 162.829]
  Call Extruder(502.66463)
  MoveL 214 to (528.35, 538.13, 4) mm, rotated rx -180 ry 0 rz 160 deg; joints [10.333, 84.728, -26.011, -145.602, 63.373, 162.941]
  Call Extruder(504.40968)
  MoveL 215 to (527.6, 538.67, 4) mm, rotated rx -180 ry 0 rz 160 deg; joints [10.412, 84.606, -25.738, -145.56, 63.521, 162.998]
  Call Extruder(507.92565)
  MoveL 216 to (526.05, 539.73, 4) mm, rotated rx -180 ry 0 rz 160 deg; joints [10.568, 84.356, -25.176, -145.481, 63.823, 163.122]
  Call Extruder(510.68628)
  MoveL 217 to (524.81, 540.51, 4) mm, rotated rx -180 ry 0 rz 160 deg; joints [10.687, 84.156, -24.725, -145.424, 64.064, 163.225]
  Call Extruder(511.74634)
  MoveL 218 to (524.33, 540.8, 4) mm, rotated rx 180 ry 0 rz 160 deg; joints [10.731, 84.078, -24.55, -145.403, 64.157, 163.265]
  Call Extruder(515.29928)
  MoveL 219 to (522.69, 541.74, 4) mm, rotated rx 180 ry 0 rz 160 deg; joints [10.878, 83.816, -23.956, -145.338, 64.472, 163.407]
  Call Extruder(516.74405)
  MoveL 220 to (522.01, 542.1, 4) mm, rotated rx -180 ry 0 rz 160 deg; joints [10.935, 83.707, -23.71, -145.315, 64.601, 163.468]
  Call Extruder(519.52351)
  MoveL 221 to (520.69, 542.76, 4) mm, rotated rx -180 ry 0 rz 160 deg; joints [11.043, 83.497, -23.233, -145.272, 64.852, 163.587]
  Call Extruder(520.61741)
  MoveL 222 to (520.16, 543.01, 4) mm, rotated rx 180 ry 0 rz 160 deg; joints [11.084, 83.413, -23.043, -145.257, 64.951, 163.635]
  Call Extruder(523.39314)
  MoveL 223 to (518.82, 543.62, 4) mm, rotated rx -180 ry 0 rz 160 deg; joints [11.187, 83.2, -22.558, -145.22, 65.203, 163.761]
  Call Extruder(524.45597)
  MoveL 224 to (518.3, 543.84, 4) mm, rotated rx -180 ry 0 rz 160 deg; joints [11.225, 83.118, -22.37, -145.207, 65.3, 163.81]
  Call Extruder(527.27870)
  MoveL 225 to (516.9, 544.39, 4) mm, rotated rx -180 ry 0 rz 160 deg; joints [11.323, 82.899, -21.868, -145.178, 65.56, 163.944]
  Call Extruder(529.43962)
  MoveL 226 to (515.83, 544.79, 4) mm, rotated rx 180 ry 0 rz 160 deg; joints [11.396, 82.73, -21.481, -145.157, 65.759, 164.05]
  Call Extruder(532.27167)
  MoveL 227 to (514.4, 545.27, 4) mm, rotated rx -180 ry 0 rz 160 deg; joints [11.487, 82.508, -20.969, -145.135, 66.021, 164.191]
  Call Extruder(533.30864)
  MoveL 228 to (513.87, 545.43, 4) mm, rotated rx -180 ry 0 rz 160 deg; joints [11.519, 82.426, -20.781, -145.128, 66.117, 164.244]
  Call Extruder(535.78449)
  MoveL 229 to (512.61, 545.8, 4) mm, rotated rx -180 ry 0 rz 160 deg; joints [11.594, 82.23, -20.329, -145.115, 66.348, 164.373]
  Call Extruder(537.97742)
  MoveL 230 to (511.48, 546.1, 4) mm, rotated rx -180 ry 0 rz 160 deg; joints [11.657, 82.057, -19.928, -145.105, 66.552, 164.488]
  Call Extruder(538.00272)
  MoveL 231 to (511.47, 546.1, 4) mm, rotated rx 180 ry 0 rz 160 deg; joints [11.656, 82.055, -19.923, -145.106, 66.554, 164.49]
  Call Extruder(539.98190)
  MoveL 232 to (510.45, 546.34, 4) mm, rotated rx 180 ry 0 rz 160 deg; joints [11.711, 81.898, -19.559, -145.1, 66.738, 164.597]
  Call Extruder(542.21981)
  MoveL 233 to (509.29, 546.59, 4) mm, rotated rx 180 ry 0 rz 160 deg; joints [11.769, 81.719, -19.144, -145.097, 66.947, 164.719]
  Call Extruder(544.32854)
  MoveL 234 to (508.19, 546.8, 4) mm, rotated rx 180 ry 0 rz 160 deg; joints [11.822, 81.552, -18.754, -145.095, 67.144, 164.836]
  Call Extruder(546.08723)
  MoveL 235 to (507.26, 546.95, 4) mm, rotated rx -180 ry 0 rz 160 deg; joints [11.863, 81.412, -18.426, -145.097, 67.308, 164.936]
  Call Extruder(547.66448)
  MoveL 236 to (506.43, 547.07, 4) mm, rotated rx 180 ry 0 rz 160 deg; joints [11.899, 81.286, -18.132, -145.1, 67.456, 165.026]
  Call Extruder(549.87491)
  MoveL 237 to (505.27, 547.21, 4) mm, rotated rx -180 ry 0 rz 160 deg; joints [11.946, 81.11, -17.719, -145.107, 67.662, 165.154]
  Call Extruder(553.79188)
  MoveL 238 to (503.19, 547.4, 4) mm, rotated rx 180 ry 0 rz 160 deg; joints [12.022, 80.799, -16.987, -145.126, 68.027, 165.384]
  Call Extruder(557.68404)
  MoveL 239 to (501.13, 547.49, 4) mm, rotated rx -180 ry 0 rz 160 deg; joints [12.087, 80.491, -16.259, -145.154, 68.388, 165.618]
  Call Extruder(561.48380)
  MoveL 240 to (499.11, 547.5, 4) mm, rotated rx 180 ry 0 rz 160 deg; joints [12.14, 80.192, -15.549, -145.19, 68.738, 165.849]
  Set speed (60.0 mm/s)
  MoveL 241 to (501.13, 547.49, 4) mm, rotated rx -180 ry 0 rz 160 deg; joints [12.087, 80.491, -16.259, -145.154, 68.388, 165.618]
  Set speed (1000.0 mm/s)
  MoveL 242 to (503.19, 547.4, 4) mm, rotated rx 180 ry 0 rz 160 deg; joints [12.022, 80.799, -16.987, -145.126, 68.027, 165.384]
  Set speed (60.0 mm/s)
  Set speed (1000.0 mm/s)
  MoveL 243 to (505.27, 547.21, 4) mm, rotated rx -180 ry 0 rz 160 deg; joints [11.946, 81.11, -17.719, -145.107, 67.662, 165.154]
  Set speed (60.0 mm/s)
  Set speed (1000.0 mm/s)
  MoveL 244 to (506.43, 547.07, 4) mm, rotated rx 180 ry 0 rz 160 deg; joints [11.899, 81.286, -18.132, -145.1, 67.456, 165.026]
  Set speed (60.0 mm/s)
  Set speed (1000.0 mm/s)
  MoveL 245 to (507.26, 546.95, 4) mm, rotated rx -180 ry 0 rz 160 deg; joints [11.863, 81.412, -18.426, -145.097, 67.308, 164.936]
  Set speed (60.0 mm/s)
  Set speed (1000.0 mm/s)
  MoveL 246 to (508.19, 546.8, 4) mm, rotated rx 180 ry 0 rz 160 deg; joints [11.822, 81.552, -18.754, -145.095, 67.144, 164.836]
  Set speed (60.0 mm/s)
  Set speed (1000.0 mm/s)
  MoveL 247 to (509.29, 546.59, 4) mm, rotated rx 180 ry 0 rz 160 deg; joints [11.769, 81.719, -19.144, -145.097, 66.947, 164.719]
  Set speed (60.0 mm/s)
  Set speed (1000.0 mm/s)
  MoveL 248 to (510.45, 546.34, 4) mm, rotated rx 180 ry 0 rz 160 deg; joints [11.711, 81.898, -19.559, -145.1, 66.738, 164.597]
  Set speed (60.0 mm/s)
  Set speed (1000.0 mm/s)
  MoveL 249 to (511, 546.21, 4) mm, rotated rx -180 ry 0 rz 160 deg; joints [11.681, 81.983, -19.756, -145.103, 66.638, 164.539]
  Set speed (60.0 mm/s)
  Set speed (25.0 mm/s)
  Call Extruder(554.98380)
  MoveL 250 to (511, 546.21, 4) mm, rotated rx -180 ry 0 rz 160 deg; joints [11.681, 81.983, -19.756, -145.103, 66.638, 164.539]
  Set speed (60.0 mm/s)
  MoveL 251 to (499.17, 544.65, 4) mm, rotated rx 180 ry 0 rz 160 deg; joints [11.79, 80.113, -15.362, -145.579, 68.743, 166.048]
  Set speed (25.0 mm/s)
  Call Extruder(561.48380)
  MoveL 252 to (499.17, 544.65, 4) mm, rotated rx 180 ry 0 rz 160 deg; joints [11.79, 80.113, -15.362, -145.579, 68.743, 166.048]
  Set speed (30.0 mm/s)
  Call Extruder(565.27937)
  MoveL 253 to (497.16, 544.56, 4) mm, rotated rx -180 ry 0 rz 160 deg; joints [11.831, 79.818, -14.656, -145.626, 69.092, 166.281]
  Call Extruder(566.61021)
  MoveL 254 to (496.45, 544.52, 4) mm, rotated rx 180 ry 0 rz 160 deg; joints [11.844, 79.715, -14.409, -145.644, 69.213, 166.363]
  Call Extruder(568.77171)
  MoveL 255 to (495.31, 544.41, 4) mm, rotated rx -180 ry 0 rz 160 deg; joints [11.86, 79.549, -14.009, -145.676, 69.41, 166.498]
  Call Extruder(570.88560)
  MoveL 256 to (494.19, 544.28, 4) mm, rotated rx 180 ry 0 rz 160 deg; joints [11.873, 79.387, -13.62, -145.711, 69.601, 166.631]
  Call Extruder(572.36388)
  MoveL 257 to (493.41, 544.16, 4) mm, rotated rx -180 ry 0 rz 160 deg; joints [11.879, 79.275, -13.348, -145.738, 69.734, 166.724]
  Call Extruder(574.49581)
  MoveL 258 to (492.3, 543.98, 4) mm, rotated rx -180 ry 0 rz 160 deg; joints [11.885, 79.114, -12.958, -145.779, 69.925, 166.859]
  Call Extruder(578.20778)
  MoveL 259 to (490.36, 543.6, 4) mm, rotated rx 180 ry 0 rz 160 deg; joints [11.889, 78.836, -12.283, -145.856, 70.254, 167.095]
  Call Extruder(581.73033)
  MoveL 260 to (488.54, 543.16, 4) mm, rotated rx -180 ry 0 rz 160 deg; joints [11.881, 78.576, -11.649, -145.938, 70.563, 167.321]
  Call Extruder(584.99062)
  MoveL 261 to (486.87, 542.69, 4) mm, rotated rx 180 ry 0 rz 160 deg; joints [11.866, 78.34, -11.069, -146.021, 70.844, 167.53]
  Call Extruder(588.27181)
  MoveL 262 to (485.22, 542.13, 4) mm, rotated rx 180 ry 0 rz 160 deg; joints [11.839, 78.106, -10.492, -146.115, 71.123, 167.741]
  Call Extruder(588.31095)
  MoveL 263 to (485.2, 542.14, 4) mm, rotated rx 180 ry 0 rz 160 deg; joints [11.841, 78.104, -10.487, -146.114, 71.125, 167.742]
  Call Extruder(590.07138)
  MoveL 264 to (484.32, 541.81, 4) mm, rotated rx 180 ry 0 rz 160 deg; joints [11.824, 77.98, -10.181, -146.166, 71.273, 167.855]
  Call Extruder(592.73729)
  MoveL 265 to (483.01, 541.29, 4) mm, rotated rx 180 ry 0 rz 160 deg; joints [11.792, 77.795, -9.722, -146.25, 71.495, 168.026]
  Call Extruder(593.74090)
  MoveL 266 to (482.51, 541.09, 4) mm, rotated rx 180 ry 0 rz 160 deg; joints [11.78, 77.726, -9.55, -146.282, 71.577, 168.091]
  Call Extruder(596.27958)
  MoveL 267 to (481.28, 540.54, 4) mm, rotated rx -180 ry 0 rz 160 deg; joints [11.742, 77.553, -9.12, -146.368, 71.784, 168.253]
  Call Extruder(597.63000)
  MoveL 268 to (480.63, 540.23, 4) mm, rotated rx 180 ry 0 rz 160 deg; joints [11.72, 77.463, -8.894, -146.416, 71.892, 168.339]
  Call Extruder(597.67795)
  MoveL 269 to (480.61, 540.23, 4) mm, rotated rx 180 ry 0 rz 160 deg; joints [11.721, 77.46, -8.886, -146.415, 71.896, 168.342]
  Call Extruder(601.08512)
  MoveL 270 to (479, 539.41, 4) mm, rotated rx 180 ry 0 rz 160 deg; joints [11.658, 77.235, -8.323, -146.541, 72.166, 168.558]
  Call Extruder(602.22562)
  MoveL 271 to (478.46, 539.12, 4) mm, rotated rx -180 ry 0 rz 160 deg; joints [11.635, 77.161, -8.137, -146.584, 72.255, 168.63]
  Call Extruder(605.70490)
  MoveL 272 to (476.86, 538.19, 4) mm, rotated rx -180 ry 0 rz 160 deg; joints [11.558, 76.939, -7.576, -146.723, 72.523, 168.85]
  Call Extruder(608.86984)
  MoveL 273 to (475.44, 537.3, 4) mm, rotated rx 180 ry 0 rz 160 deg; joints [11.48, 76.742, -7.077, -146.855, 72.761, 169.047]
  Call Extruder(611.87534)
  MoveL 274 to (474.12, 536.39, 4) mm, rotated rx -180 ry 0 rz 160 deg; joints [11.396, 76.56, -6.615, -146.988, 72.98, 169.233]
  Call Extruder(614.00182)
  MoveL 275 to (473.21, 535.72, 4) mm, rotated rx 180 ry 0 rz 160 deg; joints [11.333, 76.435, -6.293, -147.085, 73.133, 169.363]
  Call Extruder(616.67021)
  MoveL 276 to (472.09, 534.85, 4) mm, rotated rx 180 ry 0 rz 160 deg; joints [11.249, 76.28, -5.897, -147.211, 73.32, 169.525]
  Call Extruder(617.63231)
  MoveL 277 to (471.69, 534.53, 4) mm, rotated rx 180 ry 0 rz 160 deg; joints [11.218, 76.225, -5.756, -147.257, 73.387, 169.582]
  Call Extruder(620.70773)
  MoveL 278 to (470.44, 533.48, 4) mm, rotated rx 180 ry 0 rz 160 deg; joints [11.112, 76.054, -5.314, -147.409, 73.596, 169.766]
  Call Extruder(623.91434)
  MoveL 279 to (469.19, 532.32, 4) mm, rotated rx -180 ry 0 rz 160 deg; joints [10.991, 75.881, -4.868, -147.576, 73.805, 169.954]
  Call Extruder(625.96288)
  MoveL 280 to (468.41, 531.56, 4) mm, rotated rx 180 ry 0 rz 160 deg; joints [10.911, 75.774, -4.589, -147.685, 73.936, 170.072]
  Call Extruder(628.51827)
  MoveL 281 to (467.46, 530.59, 4) mm, rotated rx 180 ry 0 rz 160 deg; joints [10.806, 75.643, -4.25, -147.824, 74.095, 170.218]
  Call Extruder(631.95177)
  MoveL 282 to (466.24, 529.23, 4) mm, rotated rx -180 ry 0 rz 160 deg; joints [10.657, 75.475, -3.809, -148.018, 74.3, 170.409]
  Call Extruder(633.21411)
  MoveL 283 to (465.8, 528.72, 4) mm, rotated rx -180 ry 0 rz 160 deg; joints [10.599, 75.415, -3.651, -148.091, 74.374, 170.479]
  Call Extruder(635.78821)
  MoveL 284 to (464.94, 527.66, 4) mm, rotated rx 180 ry 0 rz 160 deg; joints [10.479, 75.295, -3.337, -148.243, 74.519, 170.618]
  Call Extruder(637.89736)
  MoveL 285 to (464.26, 526.77, 4) mm, rotated rx 180 ry 0 rz 160 deg; joints [10.377, 75.2, -3.088, -148.37, 74.634, 170.731]
  Call Extruder(641.26840)
  MoveL 286 to (463.21, 525.32, 4) mm, rotated rx 180 ry 0 rz 160 deg; joints [10.207, 75.054, -2.702, -148.578, 74.812, 170.906]
  Call Extruder(644.18583)
  MoveL 287 to (462.36, 524.02, 4) mm, rotated rx -180 ry 0 rz 160 deg; joints [10.053, 74.934, -2.383, -148.763, 74.957, 171.054]
  Call Extruder(645.16745)
  MoveL 288 to (462.08, 523.58, 4) mm, rotated rx 180 ry 0 rz 160 deg; joints [10, 74.895, -2.279, -148.826, 75.004, 171.103]
  Call Extruder(647.40338)
  MoveL 289 to (461.46, 522.56, 4) mm, rotated rx -180 ry 0 rz 160 deg; joints [9.877, 74.809, -2.049, -148.972, 75.109, 171.213]
  Call Extruder(648.78137)
  MoveL 290 to (461.1, 521.93, 4) mm, rotated rx 180 ry 0 rz 160 deg; joints [9.8, 74.757, -1.91, -149.063, 75.171, 171.279]
  Call Extruder(651.42252)
  MoveL 291 to (460.43, 520.69, 4) mm, rotated rx 180 ry 0 rz 160 deg; joints [9.648, 74.661, -1.654, -149.24, 75.286, 171.404]
  Call Extruder(653.47012)
  MoveL 292 to (459.94, 519.72, 4) mm, rotated rx -180 ry 0 rz 160 deg; joints [9.527, 74.59, -1.464, -149.38, 75.37, 171.498]
  Call Extruder(655.70900)
  MoveL 293 to (459.43, 518.65, 4) mm, rotated rx -180 ry 0 rz 160 deg; joints [9.392, 74.516, -1.264, -149.534, 75.459, 171.598]
  Call Extruder(657.08800)
  MoveL 294 to (459.12, 517.98, 4) mm, rotated rx -180 ry 0 rz 160 deg; joints [9.308, 74.472, -1.146, -149.63, 75.511, 171.659]
  Call Extruder(660.19451)
  MoveL 295 to (458.48, 516.46, 4) mm, rotated rx -180 ry 0 rz 160 deg; joints [9.114, 74.377, -0.89, -149.849, 75.622, 171.792]
  Call Extruder(664.41844)
  MoveL 296 to (457.71, 514.35, 4) mm, rotated rx -180 ry 0 rz 160 deg; joints [8.841, 74.259, -0.573, -150.153, 75.756, 171.964]
  Call Extruder(666.99780)
  MoveL 297 to (457.29, 513.04, 4) mm, rotated rx 180 ry 0 rz 160 deg; joints [8.671, 74.194, -0.395, -150.342, 75.83, 172.064]
  Call Extruder(669.90802)
  MoveL 298 to (456.86, 511.56, 4) mm, rotated rx 180 ry 0 rz 160 deg; joints [8.475, 74.125, -0.207, -150.556, 75.907, 172.174]
  Call Extruder(669.94415)
  MoveL 299 to (456.87, 511.54, 4) mm, rotated rx 180 ry 0 rz 160 deg; joints [8.473, 74.126, -0.209, -150.558, 75.905, 172.173]
  Call Extruder(671.71856)
  MoveL 300 to (456.63, 510.63, 4) mm, rotated rx 180 ry 0 rz 160 deg; joints [8.351, 74.086, -0.102, -150.69, 75.948, 172.238]
  Call Extruder(675.29540)
  MoveL 301 to (456.22, 508.77, 4) mm, rotated rx -180 ry 0 rz 160 deg; joints [8.103, 74.015, 0.091, -150.959, 76.021, 172.361]
  Call Extruder(677.44179)
  MoveL 302 to (456, 507.65, 4) mm, rotated rx -180 ry 0 rz 160 deg; joints [7.952, 73.977, 0.197, -151.122, 76.06, 172.431]
  Call Extruder(678.94039)
  MoveL 303 to (455.88, 506.87, 4) mm, rotated rx 180 ry 0 rz 160 deg; joints [7.845, 73.952, 0.265, -151.236, 76.083, 172.479]
  Call Extruder(681.06271)
  MoveL 304 to (455.72, 505.75, 4) mm, rotated rx -180 ry 0 rz 160 deg; joints [7.693, 73.919, 0.353, -151.398, 76.113, 172.544]
  Call Extruder(682.54474)
  MoveL 305 to (455.62, 504.97, 4) mm, rotated rx 180 ry 0 rz 160 deg; joints [7.586, 73.899, 0.41, -151.511, 76.131, 172.588]
  Call Extruder(684.64257)
  MoveL 306 to (455.51, 503.86, 4) mm, rotated rx -180 ry 0 rz 160 deg; joints [7.434, 73.872, 0.483, -151.672, 76.152, 172.648]
  Call Extruder(688.24119)
  MoveL 307 to (455.39, 501.95, 4) mm, rotated rx 180 ry 0 rz 160 deg; joints [7.17, 73.834, 0.587, -151.949, 76.177, 172.745]
  Call Extruder(691.85950)
  MoveL 308 to (455.34, 500.03, 4) mm, rotated rx 180 ry 0 rz 160 deg; joints [6.903, 73.805, 0.668, -152.228, 76.189, 172.835]
  Call Extruder(695.37232)
  MoveL 309 to (455.38, 498.16, 4) mm, rotated rx 180 ry 0 rz 160 deg; joints [6.641, 73.786, 0.719, -152.499, 76.185, 172.914]
  Call Extruder(698.75879)
  MoveL 310 to (455.49, 496.36, 4) mm, rotated rx -180 ry 0 rz 160 deg; joints [6.388, 73.776, 0.746, -152.76, 76.169, 172.984]
  Call Extruder(700.97460)
  MoveL 311 to (455.6, 495.19, 4) mm, rotated rx -180 ry 0 rz 160 deg; joints [6.223, 73.774, 0.752, -152.929, 76.153, 173.026]
  Call Extruder(703.97880)
  MoveL 312 to (455.8, 493.61, 4) mm, rotated rx 180 ry 0 rz 160 deg; joints [5.998, 73.778, 0.742, -153.158, 76.12, 173.078]
  Call Extruder(707.54222)
  MoveL 313 to (456.12, 491.74, 4) mm, rotated rx 180 ry 0 rz 160 deg; joints [5.732, 73.79, 0.707, -153.428, 76.068, 173.133]
  Call Extruder(710.89969)
  MoveL 314 to (456.48, 489.99, 4) mm, rotated rx 180 ry 0 rz 160 deg; joints [5.483, 73.81, 0.654, -153.679, 76.008, 173.179]
  Call Extruder(713.10239)
  MoveL 315 to (456.76, 488.85, 4) mm, rotated rx 180 ry 0 rz 160 deg; joints [5.32, 73.827, 0.606, -153.843, 75.961, 173.206]
  Call Extruder(716.18856)
  MoveL 316 to (457.2, 487.27, 4) mm, rotated rx 180 ry 0 rz 160 deg; joints [5.093, 73.858, 0.521, -154.069, 75.886, 173.238]
  Call Extruder(719.58537)
  MoveL 317 to (457.75, 485.55, 4) mm, rotated rx 180 ry 0 rz 160 deg; joints [4.846, 73.9, 0.407, -154.314, 75.791, 173.267]
  Call Extruder(723.10828)
  MoveL 318 to (458.39, 483.79, 4) mm, rotated rx -180 ry 0 rz 160 deg; joints [4.593, 73.952, 0.264, -154.563, 75.68, 173.291]
  Call Extruder(726.48829)
  MoveL 319 to (459.07, 482.13, 4) mm, rotated rx -180 ry 0 rz 160 deg; joints [4.353, 74.01, 0.106, -154.798, 75.562, 173.307]
  Call Extruder(728.34973)
  MoveL 320 to (459.48, 481.23, 4) mm, rotated rx 180 ry 0 rz 160 deg; joints [4.223, 74.046, 0.008, -154.925, 75.491, 173.314]
  Call Extruder(729.89198)
  MoveL 321 to (459.83, 480.49, 4) mm, rotated rx 180 ry 0 rz 160 deg; joints [4.117, 74.077, -0.078, -155.028, 75.429, 173.317]
  Call Extruder(732.01948)
  MoveL 322 to (460.33, 479.47, 4) mm, rotated rx -180 ry 0 rz 160 deg; joints [3.97, 74.123, -0.201, -155.169, 75.341, 173.321]
  Call Extruder(732.07403)
  MoveL 323 to (460.36, 479.45, 4) mm, rotated rx 180 ry 0 rz 160 deg; joints [3.967, 74.125, -0.207, -155.172, 75.337, 173.32]
  Call Extruder(734.92222)
  MoveL 324 to (461.08, 478.12, 4) mm, rotated rx -180 ry 0 rz 160 deg; joints [3.775, 74.191, -0.388, -155.357, 75.211, 173.321]
  Call Extruder(734.94667)
  MoveL 325 to (461.08, 478.11, 4) mm, rotated rx -180 ry 0 rz 160 deg; joints [3.774, 74.191, -0.388, -155.359, 75.211, 173.321]
  Call Extruder(738.60921)
  MoveL 326 to (462.07, 476.43, 4) mm, rotated rx -180 ry 0 rz 160 deg; joints [3.532, 74.286, -0.644, -155.589, 75.036, 173.316]
  Call Extruder(742.02345)
  MoveL 327 to (463.06, 474.91, 4) mm, rotated rx -180 ry 0 rz 160 deg; joints [3.313, 74.382, -0.906, -155.796, 74.86, 173.304]
  Call Extruder(743.95065)
  MoveL 328 to (463.65, 474.07, 4) mm, rotated rx -180 ry 0 rz 160 deg; joints [3.192, 74.441, -1.063, -155.909, 74.755, 173.295]
  Call Extruder(745.50540)
  MoveL 329 to (464.13, 473.4, 4) mm, rotated rx 180 ry 0 rz 160 deg; joints [3.096, 74.489, -1.193, -155.999, 74.669, 173.286]
  Call Extruder(747.28866)
  MoveL 330 to (464.7, 472.65, 4) mm, rotated rx 180 ry 0 rz 160 deg; joints [2.987, 74.547, -1.349, -156.1, 74.567, 173.275]
  Call Extruder(750.84685)
  MoveL 331 to (465.89, 471.18, 4) mm, rotated rx -180 ry 0 rz 160 deg; joints [2.776, 74.669, -1.675, -156.295, 74.355, 173.247]
  Call Extruder(754.19875)
  MoveL 332 to (467.07, 469.84, 4) mm, rotated rx -180 ry 0 rz 160 deg; joints [2.585, 74.792, -2.004, -156.469, 74.144, 173.215]
  Call Extruder(756.08301)
  MoveL 333 to (467.76, 469.11, 4) mm, rotated rx -180 ry 0 rz 160 deg; joints [2.481, 74.864, -2.197, -156.563, 74.021, 173.195]
  Call Extruder(757.60079)
  MoveL 334 to (468.32, 468.53, 4) mm, rotated rx 180 ry 0 rz 160 deg; joints [2.398, 74.924, -2.357, -156.637, 73.92, 173.177]
  Call Extruder(759.50694)
  MoveL 335 to (469.04, 467.82, 4) mm, rotated rx -180 ry 0 rz 160 deg; joints [2.297, 75.002, -2.563, -156.727, 73.79, 173.153]
  Call Extruder(762.95852)
  MoveL 336 to (470.39, 466.58, 4) mm, rotated rx -180 ry 0 rz 160 deg; joints [2.12, 75.148, -2.95, -156.882, 73.547, 173.106]
  Call Extruder(766.30562)
  MoveL 337 to (471.74, 465.42, 4) mm, rotated rx 180 ry 0 rz 160 deg; joints [1.956, 75.297, -3.343, -157.024, 73.303, 173.055]
  Call Extruder(769.82859)
  MoveL 338 to (473.22, 464.27, 4) mm, rotated rx 180 ry 0 rz 160 deg; joints [1.793, 75.463, -3.777, -157.161, 73.036, 172.994]
  Call Extruder(771.68568)
  MoveL 339 to (474.02, 463.69, 4) mm, rotated rx -180 ry 0 rz 160 deg; joints [1.711, 75.553, -4.012, -157.229, 72.892, 172.96]
  Call Extruder(773.22470)
  MoveL 340 to (474.69, 463.22, 4) mm, rotated rx 180 ry 0 rz 160 deg; joints [1.645, 75.629, -4.211, -157.283, 72.77, 172.931]
  Call Extruder(775.03038)
  MoveL 341 to (475.48, 462.68, 4) mm, rotated rx 180 ry 0 rz 160 deg; joints [1.569, 75.72, -4.449, -157.344, 72.626, 172.895]
  Call Extruder(778.52872)
  MoveL 342 to (477.06, 461.69, 4) mm, rotated rx -180 ry 0 rz 160 deg; joints [1.43, 75.902, -4.922, -157.453, 72.34, 172.821]
  Call Extruder(781.92907)
  MoveL 343 to (478.62, 460.79, 4) mm, rotated rx 180 ry 0 rz 160 deg; joints [1.305, 76.087, -5.399, -157.548, 72.054, 172.744]
  Call Extruder(783.83063)
  MoveL 344 to (479.52, 460.32, 4) mm, rotated rx 180 ry 0 rz 160 deg; joints [1.24, 76.193, -5.673, -157.595, 71.891, 172.698]
  Call Extruder(786.88684)
  MoveL 345 to (480.97, 459.6, 4) mm, rotated rx 180 ry 0 rz 160 deg; joints [1.139, 76.367, -6.12, -157.666, 71.626, 172.621]
  Call Extruder(788.80026)
  MoveL 346 to (481.9, 459.18, 4) mm, rotated rx 180 ry 0 rz 160 deg; joints [1.081, 76.479, -6.407, -157.705, 71.457, 172.571]
  Call Extruder(790.58728)
  MoveL 347 to (482.77, 458.8, 4) mm, rotated rx -180 ry 0 rz 160 deg; joints [1.028, 76.585, -6.678, -157.738, 71.297, 172.522]
  Call Extruder(794.04335)
  MoveL 348 to (484.48, 458.13, 4) mm, rotated rx -180 ry 0 rz 160 deg; joints [0.936, 76.796, -7.214, -157.794, 70.984, 172.423]
  Call Extruder(797.14276)
  MoveL 349 to (486.04, 457.59, 4) mm, rotated rx 180 ry 0 rz 160 deg; joints [0.861, 76.99, -7.705, -157.833, 70.699, 172.33]
  Call Extruder(797.18829)
  MoveL 350 to (486.06, 457.57, 4) mm, rotated rx -180 ry 0 rz 160 deg; joints [0.859, 76.992, -7.711, -157.835, 70.695, 172.33]
  Call Extruder(798.90708)
  MoveL 351 to (486.93, 457.3, 4) mm, rotated rx -180 ry 0 rz 160 deg; joints [0.821, 77.102, -7.988, -157.852, 70.535, 172.276]
  Call Extruder(800.90800)
  MoveL 352 to (487.95, 457, 4) mm, rotated rx 180 ry 0 rz 160 deg; joints [0.781, 77.232, -8.315, -157.868, 70.347, 172.211]
  Call Extruder(802.78383)
  MoveL 353 to (488.91, 456.74, 4) mm, rotated rx 180 ry 0 rz 160 deg; joints [0.745, 77.355, -8.624, -157.88, 70.17, 172.15]
  Call Extruder(806.26930)
  MoveL 354 to (490.72, 456.32, 4) mm, rotated rx 180 ry 0 rz 160 deg; joints [0.687, 77.588, -9.207, -157.894, 69.838, 172.03]
  Call Extruder(809.62127)
  MoveL 355 to (492.47, 455.98, 4) mm, rotated rx 180 ry 0 rz 160 deg; joints [0.641, 77.817, -9.777, -157.895, 69.515, 171.91]
  Call Extruder(813.16606)
  MoveL 356 to (494.33, 455.71, 4) mm, rotated rx -180 ry 0 rz 160 deg; joints [0.602, 78.065, -10.391, -157.884, 69.171, 171.778]
  Call Extruder(814.58999)
  MoveL 357 to (495.08, 455.61, 4) mm, rotated rx -180 ry 0 rz 160 deg; joints [0.589, 78.165, -10.639, -157.877, 69.032, 171.723]
  Call Extruder(818.35882)
  MoveL 358 to (497.08, 455.44, 4) mm, rotated rx -180 ry 0 rz 160 deg; joints [0.564, 78.436, -11.305, -157.846, 68.663, 171.573]
  Call Extruder(821.87789)
  MoveL 359 to (498.95, 455.36, 4) mm, rotated rx 180 ry 0 rz 160 deg; joints [0.551, 78.693, -11.934, -157.804, 68.316, 171.427]
  Call Extruder(825.23560)
  MoveL 360 to (500.73, 455.35, 4) mm, rotated rx 180 ry 0 rz 160 deg; joints [0.548, 78.942, -12.541, -157.753, 67.984, 171.282]
  Call Extruder(828.15301)
  MoveL 361 to (502.28, 455.4, 4) mm, rotated rx 180 ry 0 rz 160 deg; joints [0.553, 79.161, -13.073, -157.699, 67.695, 171.152]
  Call Extruder(830.53403)
  MoveL 362 to (503.55, 455.49, 4) mm, rotated rx 180 ry 0 rz 160 deg; joints [0.562, 79.342, -13.509, -157.649, 67.46, 171.043]
  Call Extruder(834.02236)
  MoveL 363 to (505.39, 455.67, 4) mm, rotated rx -180 ry 0 rz 160 deg; joints [0.584, 79.608, -14.153, -157.567, 67.115, 170.879]
  Call Extruder(837.35056)
  MoveL 364 to (507.14, 455.92, 4) mm, rotated rx -180 ry 0 rz 160 deg; joints [0.612, 79.866, -14.769, -157.477, 66.788, 170.718]
  Call Extruder(840.90797)
  MoveL 365 to (509, 456.26, 4) mm, rotated rx 180 ry 0 rz 160 deg; joints [0.653, 80.143, -15.431, -157.37, 66.439, 170.539]
  Call Extruder(844.24203)
  MoveL 366 to (510.73, 456.65, 4) mm, rotated rx 180 ry 0 rz 160 deg; joints [0.699, 80.404, -16.053, -157.259, 66.114, 170.368]
  Call Extruder(846.07658)
  MoveL 367 to (511.68, 456.9, 4) mm, rotated rx 180 ry 0 rz 160 deg; joints [0.728, 80.548, -16.395, -157.194, 65.937, 170.271]
  Call Extruder(849.59145)
  MoveL 368 to (513.47, 457.42, 4) mm, rotated rx 180 ry 0 rz 160 deg; joints [0.79, 80.826, -17.051, -157.06, 65.599, 170.082]
  Call Extruder(852.95767)
  MoveL 369 to (515.16, 458, 4) mm, rotated rx 180 ry 0 rz 160 deg; joints [0.858, 81.092, -17.678, -156.923, 65.279, 169.897]
  Call Extruder(856.43554)
  MoveL 370 to (516.89, 458.66, 4) mm, rotated rx -180 ry 0 rz 160 deg; joints [0.936, 81.367, -18.323, -156.77, 64.953, 169.701]
  Call Extruder(858.82551)
  MoveL 371 to (518.06, 459.16, 4) mm, rotated rx 180 ry 0 rz 160 deg; joints [0.995, 81.557, -18.765, -156.66, 64.731, 169.563]
  Call Extruder(861.62875)
  MoveL 372 to (519.41, 459.79, 4) mm, rotated rx 180 ry 0 rz 160 deg; joints [1.069, 81.778, -19.28, -156.524, 64.474, 169.399]
  Call Extruder(865.14182)
  MoveL 373 to (521.08, 460.63, 4) mm, rotated rx 180 ry 0 rz 160 deg; joints [1.168, 82.054, -19.922, -156.345, 64.158, 169.19]
  Call Extruder(868.56301)
  MoveL 374 to (522.66, 461.52, 4) mm, rotated rx 180 ry 0 rz 160 deg; joints [1.272, 82.322, -20.541, -156.162, 63.856, 168.983]
  Call Extruder(871.94512)
  MoveL 375 to (524.19, 462.47, 4) mm, rotated rx 180 ry 0 rz 160 deg; joints [1.382, 82.584, -21.145, -155.973, 63.565, 168.775]
  Call Extruder(873.87546)
  MoveL 376 to (525.05, 463.04, 4) mm, rotated rx 180 ry 0 rz 160 deg; joints [1.448, 82.733, -21.487, -155.862, 63.401, 168.655]
  Call Extruder(877.25309)
  MoveL 377 to (526.51, 464.07, 4) mm, rotated rx 180 ry 0 rz 160 deg; joints [1.568, 82.991, -22.08, -155.661, 63.12, 168.442]
  Call Extruder(880.74758)
  MoveL 378 to (527.99, 465.2, 4) mm, rotated rx -180 ry 0 rz 160 deg; joints [1.699, 83.255, -22.682, -155.445, 62.838, 168.219]
  Call Extruder(884.12522)
  MoveL 379 to (529.36, 466.36, 4) mm, rotated rx 180 ry 0 rz 160 deg; joints [1.833, 83.506, -23.253, -155.23, 62.575, 168.001]
  Call Extruder(885.57254)
  MoveL 380 to (529.94, 466.87, 4) mm, rotated rx 180 ry 0 rz 160 deg; joints [1.891, 83.612, -23.494, -155.136, 62.465, 167.908]
  Call Extruder(889.40329)
  MoveL 381 to (531.42, 468.27, 4) mm, rotated rx 180 ry 0 rz 160 deg; joints [2.052, 83.888, -24.121, -154.88, 62.181, 167.658]
  Call Extruder(892.01713)
  MoveL 382 to (532.39, 469.26, 4) mm, rotated rx 180 ry 0 rz 160 deg; joints [2.166, 84.073, -24.539, -154.702, 61.995, 167.487]
  Call Extruder(895.64991)
  MoveL 383 to (533.69, 470.69, 4) mm, rotated rx 180 ry 0 rz 160 deg; joints [2.33, 84.324, -25.105, -154.448, 61.746, 167.248]
  Call Extruder(897.76223)
  MoveL 384 to (534.41, 471.55, 4) mm, rotated rx -180 ry 0 rz 160 deg; joints [2.427, 84.467, -25.427, -154.299, 61.607, 167.109]
  Call Extruder(900.34128)
  MoveL 385 to (535.27, 472.61, 4) mm, rotated rx 180 ry 0 rz 160 deg; joints [2.549, 84.639, -25.812, -154.113, 61.442, 166.939]
  Call Extruder(903.98083)
  MoveL 386 to (536.42, 474.17, 4) mm, rotated rx 180 ry 0 rz 160 deg; joints [2.726, 84.872, -26.335, -153.847, 61.222, 166.7]
  Call Extruder(904.95615)
  MoveL 387 to (536.72, 474.59, 4) mm, rotated rx -180 ry 0 rz 160 deg; joints [2.774, 84.934, -26.472, -153.775, 61.165, 166.636]
  Call Extruder(908.60762)
  MoveL 388 to (537.79, 476.21, 4) mm, rotated rx 180 ry 0 rz 160 deg; joints [2.958, 85.157, -26.971, -153.503, 60.961, 166.397]
  Call Extruder(911.24585)
  MoveL 389 to (538.52, 477.41, 4) mm, rotated rx -180 ry 0 rz 160 deg; joints [3.094, 85.312, -27.316, -153.305, 60.823, 166.226]
  Call Extruder(913.24934)
  MoveL 390 to (539.05, 478.34, 4) mm, rotated rx -180 ry 0 rz 160 deg; joints [3.199, 85.426, -27.57, -153.153, 60.723, 166.097]
  Call Extruder(915.92376)
  MoveL 391 to (539.72, 479.59, 4) mm, rotated rx -180 ry 0 rz 160 deg; joints [3.341, 85.574, -27.898, -152.949, 60.597, 165.926]
  Call Extruder(917.28824)
  MoveL 392 to (540.04, 480.24, 4) mm, rotated rx 180 ry 0 rz 160 deg; joints [3.415, 85.646, -28.059, -152.844, 60.536, 165.839]
  Call Extruder(919.57325)
  MoveL 393 to (540.57, 481.33, 4) mm, rotated rx -180 ry 0 rz 160 deg; joints [3.539, 85.766, -28.324, -152.668, 60.437, 165.695]
  Call Extruder(920.51448)
  MoveL 394 to (540.77, 481.79, 4) mm, rotated rx -180 ry 0 rz 160 deg; joints [3.59, 85.813, -28.428, -152.596, 60.399, 165.636]
  Call Extruder(923.12794)
  MoveL 395 to (541.32, 483.07, 4) mm, rotated rx 180 ry 0 rz 160 deg; joints [3.735, 85.94, -28.71, -152.394, 60.298, 165.474]
  Call Extruder(926.17357)
  MoveL 396 to (541.91, 484.58, 4) mm, rotated rx 180 ry 0 rz 160 deg; joints [3.905, 86.082, -29.023, -152.159, 60.19, 165.288]
  Call Extruder(926.20593)
  MoveL 397 to (541.9, 484.59, 4) mm, rotated rx -180 ry 0 rz 160 deg; joints [3.907, 86.08, -29.019, -152.157, 60.192, 165.288]
  Call Extruder(927.89531)
  MoveL 398 to (542.21, 485.43, 4) mm, rotated rx -180 ry 0 rz 160 deg; joints [4.003, 86.155, -29.184, -152.026, 60.137, 165.187]
  Call Extruder(928.84469)
  MoveL 399 to (542.37, 485.91, 4) mm, rotated rx -180 ry 0 rz 160 deg; joints [4.057, 86.195, -29.273, -151.953, 60.107, 165.13]
  Call Extruder(931.54437)
  MoveL 400 to (542.8, 487.28, 4) mm, rotated rx -180 ry 0 rz 160 deg; joints [4.212, 86.306, -29.516, -151.744, 60.03, 164.972]
  Call Extruder(932.49807)
  MoveL 401 to (542.95, 487.77, 4) mm, rotated rx -180 ry 0 rz 160 deg; joints [4.267, 86.342, -29.597, -151.671, 60.006, 164.917]
  Call Extruder(936.12846)
  MoveL 402 to (543.43, 489.63, 4) mm, rotated rx 180 ry 0 rz 160 deg; joints [4.478, 86.474, -29.888, -151.391, 59.922, 164.711]
  Call Extruder(938.72249)
  MoveL 403 to (543.73, 490.98, 4) mm, rotated rx 180 ry 0 rz 160 deg; joints [4.631, 86.56, -30.076, -151.192, 59.872, 164.569]
  Call Extruder(941.65025)
  MoveL 404 to (544.02, 492.51, 4) mm, rotated rx 180 ry 0 rz 160 deg; joints [4.805, 86.648, -30.269, -150.969, 59.827, 164.413]
  Call Extruder(944.39569)
  MoveL 405 to (544.24, 493.95, 4) mm, rotated rx -180 ry 0 rz 160 deg; joints [4.969, 86.72, -30.428, -150.762, 59.795, 164.272]
  Call Extruder(948.18257)
  MoveL 406 to (544.47, 495.95, 4) mm, rotated rx -180 ry 0 rz 160 deg; joints [5.197, 86.805, -30.614, -150.479, 59.769, 164.087]
  Call Extruder(951.70381)
  MoveL 407 to (544.6, 497.82, 4) mm, rotated rx -180 ry 0 rz 160 deg; joints [5.411, 86.871, -30.759, -150.219, 59.76, 163.922]
  Call Extruder(955.32250)
  MoveL 408 to (544.66, 499.74, 4) mm, rotated rx -180 ry 0 rz 160 deg; joints [5.631, 86.923, -30.871, -149.956, 59.768, 163.764]
  Call Extruder(959.04960)
  MoveL 409 to (544.62, 501.72, 4) mm, rotated rx 180 ry 0 rz 160 deg; joints [5.859, 86.957, -30.947, -149.691, 59.797, 163.613]
  Call Extruder(960.63293)
  MoveL 410 to (544.58, 502.56, 4) mm, rotated rx 180 ry 0 rz 160 deg; joints [5.956, 86.968, -30.971, -149.579, 59.813, 163.551]
  Call Extruder(962.59016)
  MoveL 411 to (544.51, 503.6, 4) mm, rotated rx 180 ry 0 rz 160 deg; joints [6.076, 86.976, -30.989, -149.443, 59.839, 163.478]
  Call Extruder(965.08106)
  MoveL 412 to (544.38, 504.92, 4) mm, rotated rx -180 ry 0 rz 160 deg; joints [6.229, 86.979, -30.995, -149.273, 59.879, 163.391]
  Call Extruder(968.38418)
  MoveL 413 to (544.15, 506.66, 4) mm, rotated rx 180 ry 0 rz 160 deg; joints [6.431, 86.971, -30.978, -149.051, 59.945, 163.284]
  Call Extruder(971.93281)
  MoveL 414 to (543.83, 508.52, 4) mm, rotated rx 180 ry 0 rz 160 deg; joints [6.649, 86.948, -30.928, -148.819, 60.031, 163.18]
  Call Extruder(974.89107)
  MoveL 415 to (543.5, 510.06, 4) mm, rotated rx -180 ry 0 rz 160 deg; joints [6.829, 86.916, -30.857, -148.631, 60.117, 163.104]
  Call Extruder(974.92193)
  MoveL 416 to (543.51, 510.07, 4) mm, rotated rx 180 ry 0 rz 160 deg; joints [6.831, 86.918, -30.862, -148.629, 60.115, 163.101]
  Call Extruder(978.54942)
  MoveL 417 to (543.03, 511.94, 4) mm, rotated rx -180 ry 0 rz 160 deg; joints [7.051, 86.865, -30.745, -148.405, 60.233, 163.019]
  Call Extruder(980.27157)
  MoveL 418 to (542.77, 512.82, 4) mm, rotated rx -180 ry 0 rz 160 deg; joints [7.156, 86.833, -30.676, -148.301, 60.295, 162.984]
  Call Extruder(982.90932)
  MoveL 419 to (542.35, 514.15, 4) mm, rotated rx -180 ry 0 rz 160 deg; joints [7.315, 86.779, -30.557, -148.145, 60.397, 162.937]
  Call Extruder(983.87537)
  MoveL 420 to (542.18, 514.64, 4) mm, rotated rx 180 ry 0 rz 160 deg; joints [7.373, 86.757, -30.509, -148.089, 60.437, 162.921]
  Call Extruder(986.71158)
  MoveL 421 to (541.66, 516.06, 4) mm, rotated rx 180 ry 0 rz 160 deg; joints [7.543, 86.687, -30.355, -147.927, 60.558, 162.88]
  Call Extruder(986.76851)
  MoveL 422 to (541.67, 516.09, 4) mm, rotated rx 180 ry 0 rz 160 deg; joints [7.547, 86.689, -30.359, -147.923, 60.557, 162.877]
  Call Extruder(990.19840)
  MoveL 423 to (540.96, 517.77, 4) mm, rotated rx -180 ry 0 rz 160 deg; joints [7.751, 86.588, -30.138, -147.735, 60.719, 162.841]
  Call Extruder(992.22598)
  MoveL 424 to (540.52, 518.75, 4) mm, rotated rx 180 ry 0 rz 160 deg; joints [7.871, 86.524, -29.998, -147.627, 60.819, 162.823]
  Call Extruder(995.26570)
  MoveL 425 to (539.82, 520.21, 4) mm, rotated rx -180 ry 0 rz 160 deg; joints [8.049, 86.421, -29.77, -147.469, 60.976, 162.805]
  Call Extruder(998.50819)
  MoveL 426 to (539.01, 521.73, 4) mm, rotated rx 180 ry 0 rz 160 deg; joints [8.237, 86.298, -29.499, -147.308, 61.156, 162.797]
  Call Extruder(999.48113)
  MoveL 427 to (538.75, 522.18, 4) mm, rotated rx 180 ry 0 rz 160 deg; joints [8.293, 86.259, -29.413, -147.261, 61.212, 162.796]
  Call Extruder(1003.12423)
  MoveL 428 to (537.76, 523.84, 4) mm, rotated rx -180 ry 0 rz 160 deg; joints [8.501, 86.105, -29.074, -147.089, 61.43, 162.802]
  Call Extruder(1005.77563)
  MoveL 429 to (536.98, 525.02, 4) mm, rotated rx -180 ry 0 rz 160 deg; joints [8.65, 85.984, -28.807, -146.97, 61.596, 162.815]
  Call Extruder(1007.77668)
  MoveL 430 to (536.38, 525.89, 4) mm, rotated rx 180 ry 0 rz 160 deg; joints [8.761, 85.889, -28.597, -146.883, 61.726, 162.829]
  Call Extruder(1010.48586)
  MoveL 431 to (535.52, 527.05, 4) mm, rotated rx 180 ry 0 rz 160 deg; joints [8.91, 85.754, -28.298, -146.77, 61.907, 162.855]
  Call Extruder(1011.46818)
  MoveL 432 to (535.21, 527.47, 4) mm, rotated rx 180 ry 0 rz 160 deg; joints [8.964, 85.704, -28.187, -146.73, 61.974, 162.865]
  Call Extruder(1014.06220)
  MoveL 433 to (534.34, 528.54, 4) mm, rotated rx 180 ry 0 rz 160 deg; joints [9.104, 85.566, -27.881, -146.627, 62.155, 162.899]
  Call Extruder(1017.76056)
  MoveL 434 to (533.05, 530.02, 4) mm, rotated rx 180 ry 0 rz 160 deg; joints [9.299, 85.36, -27.423, -146.489, 62.423, 162.958]
  Call Extruder(1019.80772)
  MoveL 435 to (532.31, 530.82, 4) mm, rotated rx 180 ry 0 rz 160 deg; joints [9.406, 85.242, -27.159, -146.416, 62.575, 162.995]
  Call Extruder(1022.35766)
  MoveL 436 to (531.36, 531.79, 4) mm, rotated rx 180 ry 0 rz 160 deg; joints [9.536, 85.09, -26.821, -146.329, 62.769, 163.047]
  Call Extruder(1026.43084)
  MoveL 437 to (529.79, 533.27, 4) mm, rotated rx 180 ry 0 rz 160 deg; joints [9.74, 84.837, -26.257, -146.199, 63.087, 163.142]
  Call Extruder(1029.67817)
  MoveL 438 to (528.47, 534.4, 4) mm, rotated rx -180 ry 0 rz 160 deg; joints [9.897, 84.627, -25.785, -146.104, 63.349, 163.229]
  Call Extruder(1030.87475)
  MoveL 439 to (527.98, 534.8, 4) mm, rotated rx 180 ry 0 rz 160 deg; joints [9.954, 84.548, -25.608, -146.071, 63.447, 163.263]
  Call Extruder(1034.12304)
  MoveL 440 to (526.62, 535.86, 4) mm, rotated rx -180 ry 0 rz 160 deg; joints [10.105, 84.33, -25.118, -145.984, 63.716, 163.36]
  Call Extruder(1035.65510)
  MoveL 441 to (525.96, 536.34, 4) mm, rotated rx -180 ry 0 rz 160 deg; joints [10.175, 84.225, -24.882, -145.946, 63.845, 163.41]
  Call Extruder(1038.97229)
  MoveL 442 to (524.5, 537.33, 4) mm, rotated rx 180 ry 0 rz 160 deg; joints [10.322, 83.993, -24.357, -145.869, 64.129, 163.523]
  Call Extruder(1041.77058)
  MoveL 443 to (523.24, 538.12, 4) mm, rotated rx -180 ry 0 rz 160 deg; joints [10.442, 83.793, -23.905, -145.81, 64.372, 163.625]
  Call Extruder(1041.80464)
  MoveL 444 to (523.24, 538.14, 4) mm, rotated rx 180 ry 0 rz 160 deg; joints [10.444, 83.793, -23.905, -145.807, 64.372, 163.624]
  Call Extruder(1045.95044)
  MoveL 445 to (521.33, 539.23, 4) mm, rotated rx 180 ry 0 rz 160 deg; joints [10.614, 83.49, -23.217, -145.73, 64.738, 163.786]
  Call Extruder(1047.28412)
  MoveL 446 to (520.7, 539.56, 4) mm, rotated rx -180 ry 0 rz 160 deg; joints [10.667, 83.391, -22.991, -145.707, 64.857, 163.841]
  Call Extruder(1049.92142)
  MoveL 447 to (519.45, 540.2, 4) mm, rotated rx 180 ry 0 rz 160 deg; joints [10.769, 83.194, -22.543, -145.665, 65.094, 163.952]
  Call Extruder(1050.93282)
  MoveL 448 to (518.96, 540.43, 4) mm, rotated rx -180 ry 0 rz 160 deg; joints [10.807, 83.118, -22.369, -145.65, 65.185, 163.995]
  Call Extruder(1054.09152)
  MoveL 449 to (517.43, 541.12, 4) mm, rotated rx 180 ry 0 rz 160 deg; joints [10.924, 82.879, -21.822, -145.606, 65.471, 164.135]
  Call Extruder(1057.20944)
  MoveL 450 to (515.89, 541.73, 4) mm, rotated rx -180 ry 0 rz 160 deg; joints [11.031, 82.639, -21.271, -145.573, 65.757, 164.282]
  Call Extruder(1059.21141)
  MoveL 451 to (514.89, 542.09, 4) mm, rotated rx 180 ry 0 rz 160 deg; joints [11.098, 82.484, -20.914, -145.553, 65.941, 164.378]
  Call Extruder(1062.35578)
  MoveL 452 to (513.31, 542.63, 4) mm, rotated rx 180 ry 0 rz 160 deg; joints [11.199, 82.24, -20.351, -145.527, 66.232, 164.532]
  Call Extruder(1065.21612)
  MoveL 453 to (511.85, 543.05, 4) mm, rotated rx 180 ry 0 rz 160 deg; joints [11.284, 82.015, -19.832, -145.51, 66.497, 164.678]
  Call Extruder(1067.29951)
  MoveL 454 to (510.78, 543.34, 4) mm, rotated rx 180 ry 0 rz 160 deg; joints [11.344, 81.852, -19.452, -145.5, 66.691, 164.786]
  Call Extruder(1067.36112)
  MoveL 455 to (510.75, 543.33, 4) mm, rotated rx 180 ry 0 rz 160 deg; joints [11.344, 81.846, -19.44, -145.502, 66.697, 164.791]
  Call Extruder(1069.17831)
  MoveL 456 to (509.81, 543.56, 4) mm, rotated rx -180 ry 0 rz 160 deg; joints [11.394, 81.704, -19.107, -145.496, 66.866, 164.887]
  Call Extruder(1071.28234)
  MoveL 457 to (508.71, 543.79, 4) mm, rotated rx -180 ry 0 rz 160 deg; joints [11.448, 81.537, -18.72, -145.492, 67.063, 165.001]
  Call Extruder(1073.18668)
  MoveL 458 to (507.72, 543.99, 4) mm, rotated rx -180 ry 0 rz 160 deg; joints [11.496, 81.387, -18.369, -145.49, 67.24, 165.105]
  Call Extruder(1074.88385)
  MoveL 459 to (506.83, 544.13, 4) mm, rotated rx 180 ry 0 rz 160 deg; joints [11.535, 81.252, -18.054, -145.492, 67.399, 165.2]
  Call Extruder(1076.34484)
  MoveL 460 to (506.06, 544.24, 4) mm, rotated rx -180 ry 0 rz 160 deg; joints [11.567, 81.137, -17.782, -145.495, 67.536, 165.283]
  Call Extruder(1078.40246)
  MoveL 461 to (504.97, 544.38, 4) mm, rotated rx 180 ry 0 rz 160 deg; joints [11.611, 80.974, -17.4, -145.5, 67.728, 165.4]
  Call Extruder(1082.13960)
  MoveL 462 to (503, 544.55, 4) mm, rotated rx -180 ry 0 rz 160 deg; joints [11.681, 80.678, -16.703, -145.519, 68.076, 165.617]
  Call Extruder(1085.82463)
  MoveL 463 to (501.04, 544.64, 4) mm, rotated rx -180 ry 0 rz 160 deg; joints [11.742, 80.388, -16.015, -145.546, 68.419, 165.836]
  Call Extruder(1089.33282)
  MoveL 464 to (499.17, 544.65, 4) mm, rotated rx 180 ry 0 rz 160 deg; joints [11.79, 80.113, -15.362, -145.579, 68.743, 166.048]
  Set speed (25.0 mm/s)
  Call Extruder(1082.83282)
  MoveL 465 to (499.17, 544.65, 4) mm, rotated rx 180 ry 0 rz 160 deg; joints [11.79, 80.113, -15.362, -145.579, 68.743, 166.048]
  Set speed (60.0 mm/s)
  MoveL 466 to (496.82, 551.07, 4) mm, rotated rx -180 ry 0 rz 160 deg; joints [12.639, 79.973, -15.026, -144.74, 69.109, 165.85]
  Set speed (1000.0 mm/s)
  MoveL 467 to (493.34, 550.74, 4) mm, rotated rx -180 ry 0 rz 160 deg; joints [12.693, 79.465, -13.808, -144.837, 69.703, 166.268]
  Set speed (60.0 mm/s)
  Set speed (1000.0 mm/s)
  MoveL 468 to (490.24, 550.23, 4) mm, rotated rx -180 ry 0 rz 160 deg; joints [12.717, 79.017, -12.725, -144.946, 70.228, 166.649]
  Set speed (60.0 mm/s)
  Set speed (1000.0 mm/s)
  MoveL 469 to (486.83, 549.45, 4) mm, rotated rx -180 ry 0 rz 160 deg; joints [12.715, 78.531, -11.538, -145.09, 70.802, 167.075]
  Set speed (60.0 mm/s)
  Set speed (1000.0 mm/s)
  MoveL 470 to (484.1, 548.63, 4) mm, rotated rx -180 ry 0 rz 160 deg; joints [12.691, 78.144, -10.587, -145.226, 71.259, 167.424]
  Set speed (60.0 mm/s)
  Set speed (1000.0 mm/s)
  MoveL 471 to (480.55, 547.33, 4) mm, rotated rx -180 ry 0 rz 160 deg; joints [12.627, 77.648, -9.355, -145.431, 71.85, 167.886]
  Set speed (60.0 mm/s)
  Set speed (1000.0 mm/s)
  MoveL 472 to (477.37, 545.89, 4) mm, rotated rx 180 ry 0 rz 160 deg; joints [12.534, 77.205, -8.248, -145.648, 72.379, 168.311]
  Set speed (60.0 mm/s)
  Set speed (1000.0 mm/s)
  MoveL 473 to (474.04, 544.1, 4) mm, rotated rx 180 ry 0 rz 160 deg; joints [12.398, 76.747, -7.09, -145.911, 72.931, 168.765]
  Set speed (60.0 mm/s)
  Set speed (1000.0 mm/s)
  MoveL 474 to (477.29, 536.69, 4) mm, rotated rx -180 ry 0 rz 160 deg; joints [11.353, 76.955, -7.616, -146.93, 72.463, 168.899]
  Set speed (60.0 mm/s)
  Set speed (25.0 mm/s)
  Call Extruder(1089.33282)
  MoveL 475 to (477.29, 536.69, 4) mm, rotated rx -180 ry 0 rz 160 deg; joints [11.353, 76.955, -7.616, -146.93, 72.463, 168.899]
  Set speed (30.0 mm/s)
  Call Extruder(1126.57849)
  MoveL 476 to (463.29, 522.69, 4) mm, rotated rx 180 ry 0 rz 160 deg; joints [9.852, 75.012, -2.589, -148.952, 74.816, 171.039]
  MoveL 477 to (462.76, 522.16, 4) mm, rotated rx -180 ry 0 rz 160 deg; joints [9.793, 74.943, -2.407, -149.028, 74.904, 171.116]
  Set speed (25.0 mm/s)
  Call Extruder(1120.07849)
  MoveL 478 to (462.76, 522.16, 4) mm, rotated rx -180 ry 0 rz 160 deg; joints [9.793, 74.943, -2.407, -149.028, 74.904, 171.116]
  Set speed (60.0 mm/s)
  MoveL 479 to (459.37, 514.53, 4) mm, rotated rx -180 ry 0 rz 160 deg; joints [8.83, 74.439, -1.059, -150.125, 75.489, 171.809]
  Set speed (25.0 mm/s)
  Call Extruder(1126.57849)
  MoveL 480 to (459.37, 514.53, 4) mm, rotated rx -180 ry 0 rz 160 deg; joints [8.83, 74.439, -1.059, -150.125, 75.489, 171.809]
  Set speed (30.0 mm/s)
  Call Extruder(1196.05797)
  MoveL 481 to (485.49, 540.65, 4) mm, rotated rx 180 ry 0 rz 160 deg; joints [11.645, 78.101, -10.481, -146.317, 71.087, 167.81]
  MoveL 482 to (486.02, 541.18, 4) mm, rotated rx 180 ry 0 rz 160 deg; joints [11.698, 78.186, -10.689, -146.238, 70.996, 167.719]
  Set speed (60.0 mm/s)
  MoveL 483 to (491.36, 542.27, 4) mm, rotated rx 180 ry 0 rz 160 deg; joints [11.697, 78.935, -12.523, -146.026, 70.094, 167.078]
  Set speed (30.0 mm/s)
  Call Extruder(1285.53029)
  MoveL 484 to (457.72, 508.63, 4) mm, rotated rx -180 ry 0 rz 160 deg; joints [8.054, 74.171, -0.333, -150.976, 75.78, 172.238]
  Set speed (60.0 mm/s)
  MoveL 485 to (457, 503.67, 4) mm, rotated rx 180 ry 0 rz 160 deg; joints [7.381, 74.025, 0.065, -151.695, 75.912, 172.532]
  Set speed (30.0 mm/s)
  Call Extruder(1390.14854)
  MoveL 486 to (496.33, 543, 4) mm, rotated rx 180 ry 0 rz 160 deg; joints [11.66, 79.653, -14.259, -145.854, 69.243, 166.484]
  Set speed (60.0 mm/s)
  MoveL 487 to (500.71, 543.14, 4) mm, rotated rx -180 ry 0 rz 160 deg; joints [11.567, 80.294, -15.792, -145.757, 68.483, 165.982]
  Set speed (30.0 mm/s)
  Call Extruder(1506.81756)
  MoveL 488 to (456.86, 499.28, 4) mm, rotated rx 180 ry 0 rz 160 deg; joints [6.774, 73.953, 0.262, -152.33, 75.944, 172.743]
  Set speed (60.0 mm/s)
  MoveL 489 to (457.1, 495.28, 4) mm, rotated rx 180 ry 0 rz 160 deg; joints [6.213, 73.931, 0.323, -152.908, 75.908, 172.901]
  Set speed (30.0 mm/s)
  Call Extruder(1633.47037)
  MoveL 490 to (504.71, 542.89, 4) mm, rotated rx 180 ry 0 rz 160 deg; joints [11.438, 80.887, -17.195, -145.709, 67.781, 165.54]
  Set speed (60.0 mm/s)
  MoveL 491 to (508.39, 542.33, 4) mm, rotated rx 180 ry 0 rz 160 deg; joints [11.28, 81.44, -18.492, -145.699, 67.127, 165.15]
  Call Extruder(0.00000)
  Set speed (30.0 mm/s)
  Call Extruder(134.90479)
  MoveL 492 to (457.68, 491.62, 4) mm, rotated rx 180 ry 0 rz 160 deg; joints [5.694, 73.951, 0.267, -153.436, 75.813, 173.014]
  Set speed (60.0 mm/s)
  MoveL 493 to (458.5, 488.2, 4) mm, rotated rx -180 ry 0 rz 160 deg; joints [5.206, 74.003, 0.126, -153.926, 75.674, 173.096]
  Set speed (30.0 mm/s)
  Call Extruder(276.71816)
  MoveL 494 to (511.81, 541.5, 4) mm, rotated rx 180 ry 0 rz 160 deg; joints [11.1, 81.959, -19.701, -145.722, 66.51, 164.801]
  Set speed (60.0 mm/s)
  MoveL 495 to (515, 540.45, 4) mm, rotated rx -180 ry 0 rz 160 deg; joints [10.901, 82.449, -20.834, -145.773, 65.926, 164.491]
  Set speed (30.0 mm/s)
  Call Extruder(424.23636)
  MoveL 496 to (459.55, 485, 4) mm, rotated rx 180 ry 0 rz 160 deg; joints [4.748, 74.084, -0.095, -154.379, 75.493, 173.15]
  Set speed (60.0 mm/s)
  MoveL 497 to (460.78, 481.99, 4) mm, rotated rx -180 ry 0 rz 160 deg; joints [4.316, 74.189, -0.382, -154.802, 75.278, 173.181]
  Set speed (30.0 mm/s)
  Call Extruder(576.45516)
  MoveL 498 to (518, 539.21, 4) mm, rotated rx 180 ry 0 rz 160 deg; joints [10.685, 82.914, -21.902, -145.847, 65.369, 164.212]
  Set speed (60.0 mm/s)
  MoveL 499 to (520.82, 537.79, 4) mm, rotated rx -180 ry 0 rz 160 deg; joints [10.455, 83.355, -22.909, -145.943, 64.837, 163.965]
  Set speed (30.0 mm/s)
  Call Extruder(732.37698)
  MoveL 500 to (462.21, 479.18, 4) mm, rotated rx -180 ry 0 rz 160 deg; joints [3.912, 74.32, -0.737, -155.192, 75.027, 173.19]
  Set speed (60.0 mm/s)
  MoveL 501 to (463.8, 476.53, 4) mm, rotated rx -180 ry 0 rz 160 deg; joints [3.53, 74.473, -1.149, -155.556, 74.746, 173.18]
  Set speed (30.0 mm/s)
  Call Extruder(891.13060)
  MoveL 502 to (523.48, 536.2, 4) mm, rotated rx -180 ry 0 rz 160 deg; joints [10.211, 83.772, -23.857, -146.062, 64.329, 163.748]
  Set speed (60.0 mm/s)
  MoveL 503 to (525.97, 534.46, 4) mm, rotated rx 180 ry 0 rz 160 deg; joints [9.955, 84.167, -24.75, -146.201, 63.844, 163.559]
  Set speed (30.0 mm/s)
  Call Extruder(1051.89267)
  MoveL 504 to (465.54, 474.03, 4) mm, rotated rx -180 ry 0 rz 160 deg; joints [3.171, 74.647, -1.616, -155.892, 74.436, 173.153]
  Set speed (60.0 mm/s)
  MoveL 505 to (467.44, 471.68, 4) mm, rotated rx 180 ry 0 rz 160 deg; joints [2.836, 74.843, -2.139, -156.201, 74.096, 173.109]
  Set speed (30.0 mm/s)
  Call Extruder(1213.81992)
  MoveL 506 to (528.31, 532.55, 4) mm, rotated rx 180 ry 0 rz 160 deg; joints [9.685, 84.537, -25.584, -146.362, 63.382, 163.4]
  Set speed (60.0 mm/s)
  MoveL 507 to (530.51, 530.51, 4) mm, rotated rx 180 ry 0 rz 160 deg; joints [9.405, 84.887, -26.367, -146.542, 62.939, 163.267]
  Set speed (30.0 mm/s)
  Call Extruder(1376.15951)
  MoveL 508 to (469.49, 469.49, 4) mm, rotated rx -180 ry 0 rz 160 deg; joints [2.522, 75.06, -2.716, -156.483, 73.729, 173.049]
  Set speed (60.0 mm/s)
  MoveL 509 to (471.68, 467.44, 4) mm, rotated rx 180 ry 0 rz 160 deg; joints [2.231, 75.299, -3.348, -156.738, 73.334, 172.972]
  Set speed (30.0 mm/s)
  Call Extruder(1538.08144)
  MoveL 510 to (532.55, 528.31, 4) mm, rotated rx 180 ry 0 rz 160 deg; joints [9.111, 85.209, -27.088, -146.746, 62.522, 163.166]
  Set speed (60.0 mm/s)
  MoveL 511 to (534.46, 525.97, 4) mm, rotated rx -180 ry 0 rz 160 deg; joints [8.805, 85.509, -27.755, -146.971, 62.126, 163.093]
  Set speed (30.0 mm/s)
  Call Extruder(1698.83687)
  MoveL 512 to (474.03, 465.54, 4) mm, rotated rx 180 ry 0 rz 160 deg; joints [1.962, 75.561, -4.034, -156.967, 72.91, 172.878]
  Set speed (60.0 mm/s)
  MoveL 513 to (476.52, 463.79, 4) mm, rotated rx -180 ry 0 rz 160 deg; joints [1.715, 75.846, -4.777, -157.167, 72.458, 172.768]
  Call Extruder(0.00000)
  Set speed (30.0 mm/s)
  Call Extruder(158.76426)
  MoveL 514 to (536.2, 523.48, 4) mm, rotated rx -180 ry 0 rz 160 deg; joints [8.486, 85.78, -28.356, -147.221, 61.756, 163.052]
  Set speed (60.0 mm/s)
  MoveL 515 to (537.79, 520.82, 4) mm, rotated rx -180 ry 0 rz 160 deg; joints [8.153, 86.022, -28.892, -147.497, 61.411, 163.045]
  Set speed (30.0 mm/s)
  Call Extruder(314.69538)
  MoveL 516 to (479.18, 462.21, 4) mm, rotated rx 180 ry 0 rz 160 deg; joints [1.492, 76.157, -5.58, -157.338, 71.976, 172.639]
  Set speed (60.0 mm/s)
  MoveL 517 to (481.99, 460.78, 4) mm, rotated rx 180 ry 0 rz 160 deg; joints [1.294, 76.495, -6.447, -157.479, 71.462, 172.49]
  Set speed (30.0 mm/s)
  Call Extruder(466.91551)
  MoveL 518 to (539.21, 518, 4) mm, rotated rx 180 ry 0 rz 160 deg; joints [7.805, 86.232, -29.354, -147.803, 61.096, 163.073]
  Set speed (60.0 mm/s)
  MoveL 519 to (540.45, 515, 4) mm, rotated rx 180 ry 0 rz 160 deg; joints [7.44, 86.405, -29.735, -148.141, 60.814, 163.14]
  Set speed (30.0 mm/s)
  Call Extruder(614.44834)
  MoveL 520 to (484.99, 459.54, 4) mm, rotated rx -180 ry 0 rz 160 deg; joints [1.121, 76.863, -7.384, -157.586, 70.913, 172.319]
  Set speed (60.0 mm/s)
  MoveL 521 to (488.19, 458.49, 4) mm, rotated rx 180 ry 0 rz 160 deg; joints [0.976, 77.266, -8.4, -157.656, 70.327, 172.122]
  Set speed (30.0 mm/s)
  Call Extruder(756.27236)
  MoveL 522 to (541.5, 511.81, 4) mm, rotated rx 180 ry 0 rz 160 deg; joints [7.058, 86.539, -30.031, -148.513, 60.566, 163.249]
  Set speed (60.0 mm/s)
  MoveL 523 to (542.33, 508.39, 4) mm, rotated rx 180 ry 0 rz 160 deg; joints [6.653, 86.625, -30.22, -148.928, 60.362, 163.407]
  Set speed (30.0 mm/s)
  Call Extruder(891.16917)
  MoveL 524 to (491.62, 457.68, 4) mm, rotated rx 180 ry 0 rz 160 deg; joints [0.862, 77.708, -9.506, -157.684, 69.697, 171.894]
  Set speed (60.0 mm/s)
  MoveL 525 to (495.28, 457.1, 4) mm, rotated rx -180 ry 0 rz 160 deg; joints [0.781, 78.195, -10.712, -157.667, 69.02, 171.633]
  Set speed (30.0 mm/s)
  Call Extruder(1017.82198)
  MoveL 526 to (542.89, 504.71, 4) mm, rotated rx 180 ry 0 rz 160 deg; joints [6.223, 86.658, -30.291, -149.392, 60.207, 163.62]
  Set speed (60.0 mm/s)
  MoveL 527 to (543.14, 500.71, 4) mm, rotated rx 180 ry 0 rz 160 deg; joints [5.76, 86.62, -30.208, -149.918, 60.116, 163.901]
  Set speed (30.0 mm/s)
  Call Extruder(1134.48435)
  MoveL 528 to (499.28, 456.86, 4) mm, rotated rx 180 ry 0 rz 160 deg; joints [0.742, 78.742, -12.053, -157.59, 68.28, 171.323]
  Set speed (60.0 mm/s)
  MoveL 529 to (503.68, 457.01, 4) mm, rotated rx -180 ry 0 rz 160 deg; joints [0.754, 79.363, -13.561, -157.439, 67.462, 170.952]
  Set speed (30.0 mm/s)
  Call Extruder(1239.06004)
  MoveL 530 to (542.99, 496.32, 4) mm, rotated rx -180 ry 0 rz 160 deg; joints [5.255, 86.5, -29.944, -150.519, 60.102, 164.262]
  Set speed (60.0 mm/s)
  MoveL 531 to (542.28, 491.37, 4) mm, rotated rx 180 ry 0 rz 160 deg; joints [4.69, 86.263, -29.423, -151.226, 60.2, 164.734]
  Set speed (30.0 mm/s)
  Call Extruder(1328.57359)
  MoveL 532 to (508.63, 457.72, 4) mm, rotated rx -180 ry 0 rz 160 deg; joints [0.836, 80.09, -15.306, -157.185, 66.536, 170.492]
  MoveL 533 to (508.1, 457.19, 4) mm, rotated rx 180 ry 0 rz 160 deg; joints [0.77, 80.01, -15.115, -157.274, 66.628, 170.566]
  Set speed (25.0 mm/s)
  Call Extruder(1322.07359)
  MoveL 534 to (508.1, 457.19, 4) mm, rotated rx 180 ry 0 rz 160 deg; joints [0.77, 80.01, -15.115, -157.274, 66.628, 170.566]
  Set speed (60.0 mm/s)
  MoveL 535 to (514.51, 459.36, 4) mm, rotated rx 180 ry 0 rz 160 deg; joints [1.027, 80.993, -17.446, -156.763, 65.431, 169.878]
  Set speed (25.0 mm/s)
  Call Extruder(1328.57359)
  MoveL 536 to (514.51, 459.36, 4) mm, rotated rx 180 ry 0 rz 160 deg; joints [1.027, 80.993, -17.446, -156.763, 65.431, 169.878]
  Set speed (30.0 mm/s)
  Call Extruder(1398.03977)
  MoveL 537 to (540.63, 485.47, 4) mm, rotated rx 180 ry 0 rz 160 deg; joints [4.02, 85.833, -28.472, -152.111, 60.486, 165.387]
  MoveL 538 to (541.16, 486, 4) mm, rotated rx 180 ry 0 rz 160 deg; joints [4.077, 85.948, -28.727, -152.011, 60.377, 165.281]
  Set speed (25.0 mm/s)
  Call Extruder(1391.53977)
  MoveL 539 to (541.16, 486, 4) mm, rotated rx 180 ry 0 rz 160 deg; joints [4.077, 85.948, -28.727, -152.011, 60.377, 165.281]
  Set speed (60.0 mm/s)
  MoveL 540 to (536.7, 477.3, 4) mm, rotated rx 180 ry 0 rz 160 deg; joints [3.093, 84.956, -26.521, -153.415, 61.215, 166.452]
  Set speed (25.0 mm/s)
  Call Extruder(1398.03977)
  MoveL 541 to (536.7, 477.3, 4) mm, rotated rx 180 ry 0 rz 160 deg; joints [3.093, 84.956, -26.521, -153.415, 61.215, 166.452]
  Set speed (30.0 mm/s)
  Call Extruder(1435.22425)
  MoveL 542 to (522.72, 463.32, 4) mm, rotated rx 180 ry 0 rz 160 deg; joints [1.49, 82.339, -20.58, -155.92, 63.878, 168.868]
  MoveL 543 to (522.19, 462.79, 4) mm, rotated rx 180 ry 0 rz 160 deg; joints [1.428, 82.248, -20.37, -156.012, 63.975, 168.952]
  Set speed (25.0 mm/s)
  Call Extruder(1428.72425)
  MoveL 544 to (522.19, 462.79, 4) mm, rotated rx 180 ry 0 rz 160 deg; joints [1.428, 82.248, -20.37, -156.012, 63.975, 168.952]
  Set speed (10.0 mm/s)
  MoveL 545 to (522.19, 462.79, 8) mm, rotated rx 180 ry 0 rz 160 deg; joints [1.428, 81.486, -19.733, -155.987, 63.861, 168.896]
  Set speed (60.0 mm/s)
  MoveL 546 to (526.27, 456.09, 8) mm, rotated rx 180 ry 0 rz 160 deg; joints [0.608, 82.157, -21.272, -156.712, 62.907, 168.909]
  Set speed (1000.0 mm/s)
  MoveL 547 to (529.46, 458.17, 8) mm, rotated rx 180 ry 0 rz 160 deg; joints [0.853, 82.721, -22.557, -156.292, 62.294, 168.461]
  Set speed (60.0 mm/s)
  Set speed (1000.0 mm/s)
  MoveL 548 to (532.05, 460.11, 8) mm, rotated rx 180 ry 0 rz 160 deg; joints [1.079, 83.192, -23.624, -155.913, 61.795, 168.07]
  Set speed (60.0 mm/s)
  Set speed (1000.0 mm/s)
  MoveL 549 to (534.51, 462.22, 8) mm, rotated rx 180 ry 0 rz 160 deg; joints [1.323, 83.653, -24.66, -155.514, 61.322, 167.671]
  Set speed (60.0 mm/s)
  Set speed (1000.0 mm/s)
  MoveL 550 to (537.12, 464.78, 8) mm, rotated rx 180 ry 0 rz 160 deg; joints [1.617, 84.158, -25.791, -155.041, 60.818, 167.214]
  Set speed (60.0 mm/s)
  Set speed (1000.0 mm/s)
  MoveL 551 to (539.43, 467.39, 8) mm, rotated rx -180 ry 0 rz 160 deg; joints [1.916, 84.623, -26.827, -154.57, 60.369, 166.771]
  Set speed (60.0 mm/s)
  Set speed (1000.0 mm/s)
  MoveL 552 to (541.73, 470.39, 8) mm, rotated rx -180 ry 0 rz 160 deg; joints [2.257, 85.102, -27.888, -154.044, 59.924, 166.29]
  Set speed (60.0 mm/s)
  Set speed (1000.0 mm/s)
  MoveL 553 to (543.32, 472.77, 8) mm, rotated rx 180 ry 0 rz 160 deg; joints [2.525, 85.445, -28.644, -153.636, 59.617, 165.927]
  Set speed (60.0 mm/s)
  Set speed (1000.0 mm/s)
  MoveL 554 to (544.77, 475.23, 8) mm, rotated rx 180 ry 0 rz 160 deg; joints [2.802, 85.768, -29.355, -153.222, 59.338, 165.568]
  Set speed (60.0 mm/s)
  Set speed (1000.0 mm/s)
  MoveL 555 to (546.48, 478.59, 8) mm, rotated rx 180 ry 0 rz 160 deg; joints [3.181, 86.165, -30.225, -152.667, 59.013, 165.099]
  Set speed (60.0 mm/s)
  Set speed (1000.0 mm/s)
  MoveL 556 to (547.83, 481.82, 8) mm, rotated rx 180 ry 0 rz 160 deg; joints [3.542, 86.497, -30.949, -152.15, 58.76, 164.676]
  Set speed (60.0 mm/s)
  Set speed (1000.0 mm/s)
  MoveL 557 to (549.04, 485.4, 8) mm, rotated rx 180 ry 0 rz 160 deg; joints [3.944, 86.814, -31.638, -151.59, 58.539, 164.235]
  Set speed (60.0 mm/s)
  Set speed (1000.0 mm/s)
  MoveL 558 to (549.78, 488.16, 8) mm, rotated rx -180 ry 0 rz 160 deg; joints [4.253, 87.022, -32.09, -151.169, 58.41, 163.915]
  Set speed (60.0 mm/s)
  Set speed (1000.0 mm/s)
  MoveL 559 to (550.52, 491.87, 8) mm, rotated rx -180 ry 0 rz 160 deg; joints [4.67, 87.252, -32.588, -150.619, 58.292, 163.515]
  Set speed (60.0 mm/s)
  Set speed (1000.0 mm/s)
  MoveL 560 to (550.96, 495.33, 8) mm, rotated rx 180 ry 0 rz 160 deg; joints [5.059, 87.419, -32.95, -150.121, 58.235, 163.172]
  Set speed (60.0 mm/s)
  Set speed (1000.0 mm/s)
  MoveL 561 to (551.11, 497.54, 8) mm, rotated rx -180 ry 0 rz 160 deg; joints [5.308, 87.5, -33.125, -149.811, 58.227, 162.969]
  Set speed (60.0 mm/s)
  Set speed (1000.0 mm/s)
  MoveL 562 to (551.17, 499.75, 8) mm, rotated rx -180 ry 0 rz 160 deg; joints [5.558, 87.562, -33.259, -149.508, 58.238, 162.778]
  Set speed (60.0 mm/s)
  Set speed (1000.0 mm/s)
  MoveL 563 to (551.07, 503.24, 8) mm, rotated rx -180 ry 0 rz 160 deg; joints [5.955, 87.619, -33.38, -149.042, 58.3, 162.505]
  Set speed (60.0 mm/s)
  Set speed (1000.0 mm/s)
  MoveL 564 to (550.77, 506.37, 8) mm, rotated rx -180 ry 0 rz 160 deg; joints [6.313, 87.629, -33.401, -148.638, 58.399, 162.287]
  Set speed (60.0 mm/s)
  Set speed (1000.0 mm/s)
  MoveL 565 to (550.22, 509.81, 8) mm, rotated rx 180 ry 0 rz 160 deg; joints [6.711, 87.593, -33.324, -148.207, 58.556, 162.081]
  Set speed (60.0 mm/s)
  Set speed (1000.0 mm/s)
  MoveL 566 to (549.36, 513.5, 8) mm, rotated rx 180 ry 0 rz 160 deg; joints [7.139, 87.497, -33.118, -147.766, 58.782, 161.901]
  Set speed (60.0 mm/s)
  Set speed (1000.0 mm/s)
  MoveL 567 to (548.32, 516.84, 8) mm, rotated rx 180 ry 0 rz 160 deg; joints [7.532, 87.36, -32.821, -147.381, 59.039, 161.776]
  Set speed (60.0 mm/s)
  Set speed (1000.0 mm/s)
  MoveL 568 to (546.95, 520.35, 8) mm, rotated rx -180 ry 0 rz 160 deg; joints [7.951, 87.158, -32.385, -146.994, 59.368, 161.687]
  Set speed (60.0 mm/s)
  Set speed (1000.0 mm/s)
  MoveL 569 to (545.45, 523.51, 8) mm, rotated rx -180 ry 0 rz 160 deg; joints [8.334, 86.926, -31.881, -146.66, 59.715, 161.646]
  Set speed (60.0 mm/s)
  Set speed (1000.0 mm/s)
  MoveL 570 to (543.59, 526.8, 8) mm, rotated rx 180 ry 0 rz 160 deg; joints [8.738, 86.628, -31.234, -146.328, 60.134, 161.646]
  Set speed (60.0 mm/s)
  Set speed (1000.0 mm/s)
  MoveL 571 to (541.66, 529.72, 8) mm, rotated rx 180 ry 0 rz 160 deg; joints [9.104, 86.311, -30.543, -146.046, 60.56, 161.688]
  Set speed (60.0 mm/s)
  Set speed (1000.0 mm/s)
  MoveL 572 to (539.36, 532.71, 8) mm, rotated rx -180 ry 0 rz 160 deg; joints [9.488, 85.93, -29.709, -145.771, 61.055, 161.775]
  Set speed (60.0 mm/s)
  Set speed (1000.0 mm/s)
  MoveL 573 to (537.03, 535.32, 8) mm, rotated rx -180 ry 0 rz 160 deg; joints [9.831, 85.543, -28.86, -145.541, 61.544, 161.894]
  Set speed (60.0 mm/s)
  Set speed (1000.0 mm/s)
  MoveL 574 to (534.32, 537.96, 8) mm, rotated rx 180 ry 0 rz 160 deg; joints [10.188, 85.093, -27.868, -145.321, 62.101, 162.061]
  Set speed (60.0 mm/s)
  Set speed (1000.0 mm/s)
  MoveL 575 to (531.65, 540.21, 8) mm, rotated rx -180 ry 0 rz 160 deg; joints [10.504, 84.65, -26.886, -145.143, 62.639, 162.25]
  Set speed (60.0 mm/s)
  Set speed (1000.0 mm/s)
  MoveL 576 to (528.6, 542.44, 8) mm, rotated rx -180 ry 0 rz 160 deg; joints [10.827, 84.148, -25.769, -144.977, 63.242, 162.488]
  Set speed (60.0 mm/s)
  Set speed (1000.0 mm/s)
  MoveL 577 to (526.18, 543.97, 8) mm, rotated rx 180 ry 0 rz 160 deg; joints [11.059, 83.754, -24.888, -144.87, 63.71, 162.691]
  Set speed (60.0 mm/s)
  Set speed (1000.0 mm/s)
  MoveL 578 to (523.69, 545.36, 8) mm, rotated rx -180 ry 0 rz 160 deg; joints [11.277, 83.35, -23.981, -144.779, 64.186, 162.912]
  Set speed (60.0 mm/s)
  Set speed (1000.0 mm/s)
  MoveL 579 to (520.28, 546.98, 8) mm, rotated rx -180 ry 0 rz 160 deg; joints [11.547, 82.804, -22.746, -144.682, 64.827, 163.229]
  Set speed (60.0 mm/s)
  Set speed (1000.0 mm/s)
  MoveL 580 to (517.03, 548.26, 8) mm, rotated rx 180 ry 0 rz 160 deg; joints [11.776, 82.288, -21.572, -144.617, 65.429, 163.547]
  Set speed (60.0 mm/s)
  Set speed (1000.0 mm/s)
  MoveL 581 to (513.42, 549.38, 8) mm, rotated rx 180 ry 0 rz 160 deg; joints [11.998, 81.724, -20.28, -144.573, 66.084, 163.913]
  Set speed (60.0 mm/s)
  Set speed (1000.0 mm/s)
  MoveL 582 to (510.02, 550.18, 8) mm, rotated rx -180 ry 0 rz 160 deg; joints [12.18, 81.198, -19.068, -144.556, 66.693, 164.271]
  Set speed (60.0 mm/s)
  Set speed (1000.0 mm/s)
  MoveL 583 to (506.92, 550.7, 8) mm, rotated rx 180 ry 0 rz 160 deg; joints [12.323, 80.725, -17.969, -144.561, 67.241, 164.607]
  Set speed (60.0 mm/s)
  Set speed (1000.0 mm/s)
  MoveL 584 to (503.44, 551.06, 8) mm, rotated rx -180 ry 0 rz 160 deg; joints [12.457, 80.201, -16.745, -144.588, 67.847, 164.993]
  Set speed (60.0 mm/s)
  Set speed (1000.0 mm/s)
  MoveL 585 to (499.44, 551.16, 8) mm, rotated rx 180 ry 0 rz 160 deg; joints [12.578, 79.604, -15.338, -144.65, 68.539, 165.451]
  Set speed (60.0 mm/s)
  Set speed (1000.0 mm/s)
  MoveL 586 to (499.43, 548.93, 8) mm, rotated rx 180 ry 0 rz 160 deg; joints [12.307, 79.531, -15.164, -144.955, 68.553, 165.616]
  Set speed (60.0 mm/s)
  Call SetRPM(255.0)
  Call M_RunCode(106)
  Set speed (25.0 mm/s)
  Call Extruder(1435.22425)
  MoveL 587 to (499.43, 548.93, 8) mm, rotated rx 180 ry 0 rz 160 deg; joints [12.307, 79.531, -15.164, -144.955, 68.553, 165.616]
  Set speed (17.5 mm/s)
  Call Extruder(1442.46875)
  MoveL 588 to (497.19, 548.86, 8) mm, rotated rx 180 ry 0 rz 160 deg; joints [12.357, 79.202, -14.382, -145.004, 68.936, 165.876]
  Set speed (17.4 mm/s)
  Call Extruder(1448.96046)
  MoveL 589 to (495.19, 548.7, 8) mm, rotated rx -180 ry 0 rz 160 deg; joints [12.392, 78.91, -13.685, -145.056, 69.277, 166.112]
  Set speed (17.4 mm/s)
  Call Extruder(1455.36845)
  MoveL 590 to (493.22, 548.46, 8) mm, rotated rx 180 ry 0 rz 160 deg; joints [12.416, 78.625, -13.001, -145.117, 69.61, 166.347]
  Set speed (17.4 mm/s)
  Call Extruder(1462.44975)
  MoveL 591 to (491.06, 548.12, 8) mm, rotated rx 180 ry 0 rz 160 deg; joints [12.432, 78.314, -12.251, -145.193, 69.974, 166.609]
  Set speed (17.4 mm/s)
  Call Extruder(1468.43234)
  MoveL 592 to (489.25, 547.74, 8) mm, rotated rx -180 ry 0 rz 160 deg; joints [12.435, 78.054, -11.623, -145.266, 70.277, 166.831]
  Set speed (17.4 mm/s)
  Call Extruder(1471.60340)
  MoveL 593 to (488.3, 547.52, 8) mm, rotated rx -180 ry 0 rz 160 deg; joints [12.433, 77.919, -11.293, -145.307, 70.437, 166.949]
  Set speed (17.4 mm/s)
  Call Extruder(1475.26098)
  MoveL 594 to (487.2, 547.24, 8) mm, rotated rx -180 ry 0 rz 160 deg; joints [12.428, 77.763, -10.913, -145.357, 70.62, 167.086]
  Set speed (17.5 mm/s)
  Call Extruder(1480.41881)
  MoveL 595 to (485.67, 546.79, 8) mm, rotated rx -180 ry 0 rz 160 deg; joints [12.415, 77.546, -10.382, -145.433, 70.875, 167.28]
  Set speed (17.5 mm/s)
  Call Extruder(1482.68762)
  MoveL 596 to (485, 546.58, 8) mm, rotated rx 180 ry 0 rz 160 deg; joints [12.407, 77.451, -10.15, -145.469, 70.986, 167.365]
  Set speed (17.5 mm/s)
  Call Extruder(1487.62566)
  MoveL 597 to (483.55, 546.09, 8) mm, rotated rx 180 ry 0 rz 160 deg; joints [12.386, 77.248, -9.649, -145.548, 71.227, 167.55]
  Set speed (17.5 mm/s)
  Call Extruder(1494.70571)
  MoveL 598 to (481.51, 545.31, 8) mm, rotated rx 180 ry 0 rz 160 deg; joints [12.343, 76.961, -8.941, -145.672, 71.566, 167.815]
  Set speed (17.4 mm/s)
  Call Extruder(1499.25635)
  MoveL 599 to (480.22, 544.76, 8) mm, rotated rx -180 ry 0 rz 160 deg; joints [12.309, 76.781, -8.493, -145.757, 71.78, 167.985]
  Call Extruder(1502.14012)
  MoveL 600 to (479.41, 544.39, 8) mm, rotated rx -180 ry 0 rz 160 deg; joints [12.285, 76.668, -8.212, -145.813, 71.914, 168.092]
  Set speed (17.5 mm/s)
  Call Extruder(1507.16199)
  MoveL 601 to (478.01, 543.72, 8) mm, rotated rx -180 ry 0 rz 160 deg; joints [12.238, 76.473, -7.727, -145.915, 72.145, 168.279]
  Set speed (17.5 mm/s)
  Call Extruder(1512.14500)
  MoveL 602 to (476.64, 543, 8) mm, rotated rx 180 ry 0 rz 160 deg; joints [12.183, 76.284, -7.253, -146.022, 72.37, 168.463]
  Set speed (17.5 mm/s)
  Call Extruder(1516.31032)
  MoveL 603 to (475.52, 542.37, 8) mm, rotated rx -180 ry 0 rz 160 deg; joints [12.134, 76.129, -6.862, -146.114, 72.556, 168.617]
  Set speed (17.5 mm/s)
  Call Extruder(1518.41477)
